SPLINE
SPL {X  -162.820, Y  +438.487, Z    +0.000, E1   -25.409, E3 +468676.662}
SPL {X  -162.820, Y  +441.593, Z    +0.000, E1   -25.391, E3 +468690.270}
SPL {X  -162.820, Y  +444.317, Z    +0.000, E1   -25.492, E3 +468701.452}
SPL {X  -162.820, Y  +446.544, Z    +0.000, E1   -25.427, E3 +468711.621}
SPL {X  -162.820, Y  +448.500, Z    +0.000, E1   -25.425, E3 +468720.223}
SPL {X  -162.820, Y  +451.056, Z    +0.000, E1   -25.443, E3 +468731.330}
SPL {X  -162.820, Y  +454.662, Z    +0.000, E1   -25.474, E3 +468747.074}
SPL {X  -162.820, Y  +458.079, Z    +0.000, E1   -25.369, E3 +468762.654}
SPL {X  -162.820, Y  +460.719, Z    +0.000, E1   -25.411, E3 +468773.912}
SPL {X  -162.820, Y  +463.419, Z    +0.000, E1   -25.510, E3 +468784.949}
SPL {X  -162.820, Y  +466.458, Z    +0.000, E1   -25.433, E3 +468799.005}
SPL {X  -162.820, Y  +470.010, Z    +0.000, E1   -25.445, E3 +468814.373}
SPL {X  -162.820, Y  +472.345, Z    +0.000, E1   -25.448, E3 +468824.460}
SPL {X  -162.820, Y  +475.191, Z    +0.000, E1   -25.489, E3 +468836.822}
SPL {X  -162.820, Y  +478.461, Z    +0.000, E1   -25.410, E3 +468851.592}
SPL {X  -162.820, Y  +480.780, Z    +0.000, E1   -25.447, E3 +468861.453}
SPL {X  -162.820, Y  +483.622, Z    +0.000, E1   -25.381, E3 +468874.495}
SPL {X  -162.820, Y  +487.570, Z    +0.000, E1   -25.482, E3 +468891.133}
SPL {X  -162.820, Y  +491.017, Z    +0.000, E1   -25.445, E3 +468906.348}
SPL {X  -162.820, Y  +494.454, Z    +0.000, E1   -25.465, E3 +468921.407}
SPL {X  -162.820, Y  +498.644, Z    +0.000, E1   -25.463, E3 +468939.784}
SPL {X  -162.820, Y  +502.845, Z    +0.000, E1   -25.458, E3 +468958.217}
SPL {X  -162.820, Y  +506.050, Z    +0.000, E1   -25.420, E3 +468972.357}
SPL {X  -162.820, Y  +508.346, Z    +0.000, E1   -25.444, E3 +468982.205}
SPL {X  -162.820, Y  +511.422, Z    +0.000, E1   -25.445, E3 +468995.865}
SPL {X  -162.820, Y  +515.039, Z    +0.000, E1   -25.452, E3 +469011.547}
SPL {X  -162.820, Y  +518.350, Z    +0.000, E1   -25.425, E3 +469026.296}
SPL {X  -162.820, Y  +521.486, Z    +0.000, E1   -25.382, E3 +469040.324}
SPL {X  -162.820, Y  +524.180, Z    +0.000, E1   -25.495, E3 +469051.196}
SPL {X  -162.820, Y  +527.020, Z    +0.000, E1   -25.477, E3 +469063.889}
SPL {X  -162.820, Y  +530.432, Z    +0.000, E1   -25.477, E3 +469078.755}
SPL {X  -162.820, Y  +534.051, Z    +0.000, E1   -25.484, E3 +469094.632}
SPL {X  -162.820, Y  +537.226, Z    +0.000, E1   -25.378, E3 +469109.201}
SPL {X  -162.820, Y  +539.521, Z    +0.000, E1   -25.386, E3 +469119.160}
SPL {X  -162.820, Y  +542.667, Z    +0.000, E1   -25.474, E3 +469132.485}
SPL {X  -162.820, Y  +546.125, Z    +0.000, E1   -25.505, E3 +469147.210}
SPL {X  -162.820, Y  +549.578, Z    +0.000, E1   -25.462, E3 +469162.834}
SPL {X  -162.820, Y  +553.157, Z    +0.000, E1   -25.443, E3 +469178.497}
SPL {X  -162.820, Y  +556.965, Z    +0.000, E1   -25.478, E3 +469195.090}
SPL {X  -162.820, Y  +561.429, Z    +0.000, E1   -25.478, E3 +469214.608}
SPL {X  -162.820, Y  +565.606, Z    +0.000, E1   -25.468, E3 +469232.939}
SPL {X  -162.820, Y  +568.974, Z    +0.000, E1   -25.453, E3 +469247.649}
SPL {X  -162.820, Y  +572.331, Z    +0.000, E1   -25.489, E3 +469262.198}
SPL {X  -162.820, Y  +576.045, Z    +0.000, E1   -25.412, E3 +469279.006}
SPL {X  -162.820, Y  +580.038, Z    +0.000, E1   -25.473, E3 +469296.101}
SPL {X  -162.820, Y  +583.044, Z    +0.000, E1   -25.450, E3 +469309.224}
SPL {X  -162.820, Y  +585.512, Z    +0.000, E1   -25.448, E3 +469320.120}
SPL {X  -162.820, Y  +588.371, Z    +0.000, E1   -25.460, E3 +469332.506}
SPL {X  -162.820, Y  +591.246, Z    +0.000, E1   -25.415, E3 +469345.525}
SPL {X  -162.820, Y  +594.339, Z    +0.000, E1   -25.487, E3 +469358.428}
SPL {X  -162.820, Y  +596.868, Z    +0.000, E1   -25.461, E3 +469369.691}
SPL {X  -162.820, Y  +600.326, Z    +0.000, E1   -25.438, E3 +469385.212}
SPL {X  -162.820, Y  +604.526, Z    +0.000, E1   -25.502, E3 +469403.035}
SPL {X  -162.820, Y  +607.811, Z    +0.000, E1   -25.507, E3 +469417.250}
SPL {X  -162.820, Y  +611.438, Z    +0.000, E1   -25.467, E3 +469433.610}
SPL {X  -162.820, Y  +615.388, Z    +0.000, E1   -25.455, E3 +469450.869}
SPL {X  -162.820, Y  +618.995, Z    +0.000, E1   -25.483, E3 +469466.464}
SPL {X  -162.820, Y  +622.118, Z    +0.000, E1   -25.492, E3 +469479.929}
SPL {X  -162.820, Y  +624.430, Z    +0.000, E1   -25.475, E3 +469490.150}
SPL {X  -162.820, Y  +626.570, Z    +0.000, E1   -25.441, E3 +469499.751}
SPL {X  -162.820, Y  +628.902, Z    +0.000, E1   -25.449, E3 +469509.931}
SPL {X  -162.820, Y  +631.177, Z    +0.000, E1   -25.467, E3 +469519.762}
SPL {X  -162.820, Y  +633.994, Z    +0.000, E1   -25.503, E3 +469531.809}
SPL {X  -162.820, Y  +636.469, Z    +0.000, E1   -25.465, E3 +469542.852}
SPL {X  -162.820, Y  +638.486, Z    +0.000, E1   -25.456, E3 +469551.770}
SPL {X  -162.820, Y  +640.803, Z    +0.000, E1   -25.462, E3 +469561.831}
SPL {X  -162.820, Y  +643.028, Z    +0.000, E1   -25.494, E3 +469571.341}
SPL {X  -162.820, Y  +646.519, Z    +0.000, E1   -25.551, E3 +469586.323}
SPL {X  -162.820, Y  +649.837, Z    +0.000, E1   -25.446, E3 +469601.447}
SPL {X  -162.820, Y  +652.810, Z    +0.000, E1   -25.497, E3 +469614.090}
SPL {X  -162.820, Y  +655.214, Z    +0.000, E1   -25.485, E3 +469624.593}
SPL {X  -162.820, Y  +657.616, Z    +0.000, E1   -25.511, E3 +469634.947}
SPL {X  -162.820, Y  +660.007, Z    +0.000, E1   -25.550, E3 +469645.008}
SPL {X  -162.820, Y  +662.980, Z    +0.000, E1   -25.505, E3 +469658.567}
SPL {X  -162.820, Y  +667.253, Z    +0.000, E1   -25.483, E3 +469677.443}
SPL {X  -162.820, Y  +671.102, Z    +0.000, E1   -25.514, E3 +469693.894}
SPL {X  -162.820, Y  +673.648, Z    +0.000, E1   -25.431, E3 +469705.560}
SPL {X  -162.796, Y  +676.319, Z    +0.000, E1   -25.526, E3 +469716.570}
SPL {X  -162.707, Y  +679.552, Z    +0.000, E1   -25.443, E3 +469731.445}
SPL {X  -162.545, Y  +682.952, Z    +0.000, E1   -25.510, E3 +469745.678}
SPL {X  -162.381, Y  +685.455, Z    +0.000, E1   -25.410, E3 +469757.364}
SPL {X  -162.194, Y  +687.760, Z    +0.000, E1   -25.360, E3 +469767.800}
SPL {X  -161.866, Y  +691.104, Z    +0.000, E1   -25.383, E3 +469782.432}
SPL {X  -161.319, Y  +695.558, Z    +0.000, E1   -25.832, E3 +469798.234}
SPL {X  -157.976, Y  +712.921, Z    +0.000, E1   -33.197, E3 +469811.626}
ENDSPLINE

SPLINE
SPL {X  -160.738, Y  +699.453, Z    +0.000, E1   -21.994, E3 +469849.253}
SPL {X  -161.689, Y  +692.657, Z    +0.000, E1   -15.656, E3 +469889.323}
SPL {X  -162.807, Y  +675.545, Z    +0.000, E1    -5.787, E3 +469884.822}
ENDSPLINE

SPLINE
SPL {X  -162.791, Y  +676.574, Z    +0.000, E1    -6.127, E3 +469897.925}
ENDSPLINE

SPLINE
SPL {X  -162.820, Y  +664.716, Z    +0.000, E1    +1.705, E3 +469886.799}
SPL {X  -162.820, Y  +658.484, Z    +0.000, E1    +6.336, E3 +469893.276}
SPL {X  -162.820, Y  +640.102, Z    +0.000, E1   +22.409, E3 +469888.014}
SPL {X  -162.820, Y  +633.503, Z    +0.000, E1   +21.975, E3 +469920.251}
SPL {X  -162.820, Y  +611.299, Z    +0.000, E1   +31.088, E3 +469948.363}
ENDSPLINE

SPLINE
SPL {X  -162.820, Y  +618.877, Z    +0.000, E1   +25.259, E3 +469959.858}
ENDSPLINE

SPLINE
SPL {X  -162.820, Y  +617.582, Z    +0.000, E1   +24.552, E3 +469971.235}
SPL {X  -162.820, Y  +614.716, Z    +0.000, E1   +24.535, E3 +469984.446}
SPL {X  -162.820, Y  +611.754, Z    +0.000, E1   +24.563, E3 +469997.734}
SPL {X  -162.820, Y  +608.970, Z    +0.000, E1   +24.542, E3 +470010.574}
SPL {X  -162.820, Y  +606.285, Z    +0.000, E1   +24.533, E3 +470022.910}
SPL {X  -162.820, Y  +603.509, Z    +0.000, E1   +24.546, E3 +470035.447}
SPL {X  -162.820, Y  +600.818, Z    +0.000, E1   +24.590, E3 +470047.370}
SPL {X  -162.820, Y  +598.053, Z    +0.000, E1   +24.547, E3 +470060.353}
SPL {X  -162.820, Y  +595.188, Z    +0.000, E1   +24.538, E3 +470073.441}
SPL {X  -162.820, Y  +592.738, Z    +0.000, E1   +24.551, E3 +470084.490}
SPL {X  -162.820, Y  +590.118, Z    +0.000, E1   +24.544, E3 +470096.549}
SPL {X  -162.820, Y  +587.204, Z    +0.000, E1   +24.592, E3 +470109.426}
SPL {X  -162.820, Y  +584.766, Z    +0.000, E1   +24.499, E3 +470121.259}
SPL {X  -162.820, Y  +581.896, Z    +0.000, E1   +24.528, E3 +470134.201}
SPL {X  -162.820, Y  +579.244, Z    +0.000, E1   +24.610, E3 +470145.545}
SPL {X  -162.820, Y  +576.848, Z    +0.000, E1   +24.543, E3 +470157.086}
SPL {X  -162.820, Y  +573.694, Z    +0.000, E1   +24.535, E3 +470171.556}
SPL {X  -162.820, Y  +570.310, Z    +0.000, E1   +24.556, E3 +470186.872}
SPL {X  -162.820, Y  +567.494, Z    +0.000, E1   +24.547, E3 +470199.657}
SPL {X  -162.820, Y  +564.977, Z    +0.000, E1   +24.571, E3 +470210.987}
SPL {X  -162.820, Y  +562.356, Z    +0.000, E1   +24.575, E3 +470222.886}
SPL {X  -162.820, Y  +558.990, Z    +0.000, E1   +24.558, E3 +470238.536}
SPL {X  -162.820, Y  +555.584, Z    +0.000, E1   +24.559, E3 +470253.905}
SPL {X  -162.820, Y  +552.169, Z    +0.000, E1   +24.581, E3 +470269.474}
SPL {X  -162.820, Y  +548.172, Z    +0.000, E1   +24.564, E3 +470287.822}
SPL {X  -162.820, Y  +544.025, Z    +0.000, E1   +24.611, E3 +470306.376}
SPL {X  -162.820, Y  +540.573, Z    +0.000, E1   +24.503, E3 +470322.830}
SPL {X  -162.820, Y  +537.211, Z    +0.000, E1   +24.561, E3 +470337.759}
SPL {X  -162.820, Y  +534.025, Z    +0.000, E1   +24.589, E3 +470352.003}
SPL {X  -162.820, Y  +531.527, Z    +0.000, E1   +24.582, E3 +470363.388}
SPL {X  -162.820, Y  +529.165, Z    +0.000, E1   +24.521, E3 +470374.637}
SPL {X  -162.820, Y  +525.802, Z    +0.000, E1   +24.585, E3 +470389.657}
SPL {X  -162.820, Y  +521.731, Z    +0.000, E1   +24.542, E3 +470408.593}
SPL {X  -162.820, Y  +518.185, Z    +0.000, E1   +24.561, E3 +470424.465}
SPL {X  -162.820, Y  +508.728, Z    +0.000, E1   +28.484, E3 +470435.005}
SPL {X  -162.820, Y  +500.664, Z    +0.000, E1   +31.476, E3 +470443.669}
SPL {X  -162.820, Y  +499.290, Z    +0.000, E1   +30.657, E3 +470453.951}
SPL {X  -162.820, Y  +497.700, Z    +0.000, E1   +29.785, E3 +470465.566}
SPL {X  -162.820, Y  +495.915, Z    +0.000, E1   +28.861, E3 +470478.658}
SPL {X  -162.820, Y  +494.678, Z    +0.000, E1   +27.647, E3 +470492.004}
SPL {X  -162.820, Y  +493.757, Z    +0.000, E1   +26.462, E3 +470504.364}
SPL {X  -162.820, Y  +492.330, Z    +0.000, E1   +25.953, E3 +470514.118}
SPL {X  -162.820, Y  +489.800, Z    +0.000, E1   +25.653, E3 +470527.580}
SPL {X  -162.820, Y  +485.392, Z    +0.000, E1   +25.667, E3 +470546.607}
SPL {X  -162.820, Y  +482.092, Z    +0.000, E1   +25.593, E3 +470561.295}
SPL {X  -162.820, Y  +479.578, Z    +0.000, E1   +25.634, E3 +470571.938}
SPL {X  -162.820, Y  +477.137, Z    +0.000, E1   +25.632, E3 +470582.517}
SPL {X  -162.820, Y  +473.770, Z    +0.000, E1   +25.664, E3 +470597.063}
SPL {X  -162.820, Y  +469.694, Z    +0.000, E1   +25.657, E3 +470614.794}
SPL {X  -162.820, Y  +465.727, Z    +0.000, E1   +25.676, E3 +470631.837}
SPL {X  -162.820, Y  +461.675, Z    +0.000, E1   +25.655, E3 +470649.643}
SPL {X  -162.820, Y  +457.479, Z    +0.000, E1   +25.656, E3 +470667.823}
SPL {X  -162.820, Y  +453.678, Z    +0.000, E1   +25.652, E3 +470684.275}
SPL {X  -162.820, Y  +450.466, Z    +0.000, E1   +25.644, E3 +470698.220}
SPL {X  -162.820, Y  +447.822, Z    +0.000, E1   +25.664, E3 +470709.478}
SPL {X  -162.820, Y  +445.556, Z    +0.000, E1   +25.626, E3 +470719.609}
SPL {X  -162.820, Y  +442.508, Z    +0.000, E1   +25.657, E3 +470732.703}
SPL {X  -162.820, Y  +439.273, Z    +0.000, E1   +25.576, E3 +470747.341}
SPL {X  -162.820, Y  +435.635, Z    +0.000, E1   +25.661, E3 +470762.572}
SPL {X  -162.820, Y  +431.823, Z    +0.000, E1   +25.651, E3 +470779.221}
SPL {X  -162.820, Y  +427.740, Z    +0.000, E1   +25.667, E3 +470796.849}
SPL {X  -162.820, Y  +423.655, Z    +0.000, E1   +25.628, E3 +470814.874}
SPL {X  -162.820, Y  +419.407, Z    +0.000, E1   +25.665, E3 +470833.066}
SPL {X  -162.820, Y  +415.900, Z    +0.000, E1   +25.638, E3 +470848.335}
SPL {X  -162.820, Y  +412.302, Z    +0.000, E1   +25.662, E3 +470863.947}
SPL {X  -162.820, Y  +408.133, Z    +0.000, E1   +25.637, E3 +470882.205}
SPL {X  -162.820, Y  +404.293, Z    +0.000, E1   +25.628, E3 +470898.928}
SPL {X  -162.820, Y  +400.835, Z    +0.000, E1   +25.694, E3 +470913.327}
SPL {X  -162.820, Y  +398.703, Z    +0.000, E1   +25.586, E3 +470923.319}
SPL {X  -162.820, Y  +395.582, Z    +0.000, E1   +25.684, E3 +470936.311}
SPL {X  -162.820, Y  +391.417, Z    +0.000, E1   +25.659, E3 +470954.649}
SPL {X  -162.820, Y  +387.939, Z    +0.000, E1   +25.627, E3 +470969.796}
SPL {X  -162.820, Y  +384.398, Z    +0.000, E1   +25.707, E3 +470984.694}
SPL {X  -162.820, Y  +380.448, Z    +0.000, E1   +25.674, E3 +471002.057}
SPL {X  -162.785, Y  +377.106, Z    +0.000, E1   +25.598, E3 +471017.001}
SPL {X  -162.663, Y  +373.346, Z    +0.000, E1   +25.707, E3 +471032.652}
SPL {X  -162.487, Y  +370.088, Z    +0.000, E1   +25.525, E3 +471047.987}
SPL {X  -162.307, Y  +367.587, Z    +0.000, E1   +25.577, E3 +471058.405}
SPL {X  -162.041, Y  +364.588, Z    +0.000, E1   +25.591, E3 +471071.483}
SPL {X  -161.760, Y  +361.954, Z    +0.000, E1   +25.495, E3 +471083.430}
SPL {X  -161.454, Y  +359.455, Z    +0.000, E1   +25.428, E3 +471094.905}
SPL {X  -160.939, Y  +355.820, Z    +0.000, E1   +26.179, E3 +471104.788}
SPL {X  -155.035, Y  +330.756, Z    +0.000, E1   +37.918, E3 +471111.121}
SPL {X  -153.918, Y  +327.401, Z    +0.000, E1   +34.677, E3 +471146.422}
ENDSPLINE

SPLINE
SPL {X  -159.701, Y  +348.785, Z    +0.000, E1   +24.361, E3 +471153.903}
SPL {X  -162.442, Y  +369.407, Z    +0.000, E1   +11.234, E3 +471183.538}
SPL {X  -162.820, Y  +384.333, Z    +0.000, E1    +1.902, E3 +471184.744}
SPL {X  -162.820, Y  +389.940, Z    +0.000, E1    -2.281, E3 +471187.666}
SPL {X  -162.820, Y  +396.652, Z    +0.000, E1    -7.520, E3 +471187.244}
SPL {X  -162.820, Y  +406.605, Z    +0.000, E1   -16.760, E3 +471179.721}
SPL {X  -162.820, Y  +418.675, Z    +0.000, E1   -22.201, E3 +471205.970}
SPL {X  -162.820, Y  +425.113, Z    +0.000, E1   -25.243, E3 +471214.906}
SPL {X  -162.820, Y  +441.937, Z    +0.000, E1   -31.578, E3 +471236.984}
ENDSPLINE

SPLINE
SPL {X  -162.820, Y  +437.771, Z    +0.000, E1   -26.555, E3 +471256.084}
ENDSPLINE

SPLINE
SPL {X  -162.820, Y  +439.120, Z    +0.000, E1   -25.352, E3 +471270.628}
SPL {X  -162.820, Y  +441.593, Z    +0.000, E1   -25.391, E3 +471281.179}
SPL {X  -162.820, Y  +444.317, Z    +0.000, E1   -25.492, E3 +471292.361}
SPL {X  -162.820, Y  +446.544, Z    +0.000, E1   -25.427, E3 +471302.530}
SPL {X  -162.820, Y  +448.500, Z    +0.000, E1   -25.425, E3 +471311.132}
SPL {X  -162.820, Y  +451.056, Z    +0.000, E1   -25.443, E3 +471322.239}
SPL {X  -162.820, Y  +454.662, Z    +0.000, E1   -25.474, E3 +471337.984}
SPL {X  -162.820, Y  +458.079, Z    +0.000, E1   -25.369, E3 +471353.563}
SPL {X  -162.820, Y  +460.719, Z    +0.000, E1   -25.411, E3 +471364.821}
SPL {X  -162.820, Y  +463.419, Z    +0.000, E1   -25.510, E3 +471375.859}
SPL {X  -162.820, Y  +465.376, Z    +0.000, E1   -25.372, E3 +471385.446}
SPL {X  -162.820, Y  +467.440, Z    +0.000, E1   -25.427, E3 +471394.078}
SPL {X  -162.820, Y  +470.010, Z    +0.000, E1   -25.445, E3 +471405.283}
SPL {X  -162.820, Y  +473.445, Z    +0.000, E1   -25.493, E3 +471420.006}
SPL {X  -162.820, Y  +476.157, Z    +0.000, E1   -25.426, E3 +471432.221}
SPL {X  -162.820, Y  +478.461, Z    +0.000, E1   -25.410, E3 +471442.501}
SPL {X  -162.820, Y  +481.644, Z    +0.000, E1   -25.433, E3 +471456.447}
SPL {X  -162.820, Y  +486.042, Z    +0.000, E1   -25.483, E3 +471475.367}
SPL {X  -162.820, Y  +490.287, Z    +0.000, E1   -25.463, E3 +471494.085}
SPL {X  -162.820, Y  +494.454, Z    +0.000, E1   -25.465, E3 +471512.316}
SPL {X  -162.820, Y  +498.644, Z    +0.000, E1   -25.463, E3 +471530.693}
SPL {X  -162.820, Y  +502.845, Z    +0.000, E1   -25.458, E3 +471549.126}
SPL {X  -162.820, Y  +506.050, Z    +0.000, E1   -25.420, E3 +471563.266}
SPL {X  -162.820, Y  +508.346, Z    +0.000, E1   -25.444, E3 +471573.114}
SPL {X  -162.820, Y  +511.422, Z    +0.000, E1   -25.445, E3 +471586.775}
SPL {X  -162.820, Y  +515.039, Z    +0.000, E1   -25.452, E3 +471602.456}
SPL {X  -162.820, Y  +517.481, Z    +0.000, E1   -25.432, E3 +471613.190}
SPL {X  -162.820, Y  +519.134, Z    +0.000, E1   -25.366, E3 +471620.937}
SPL {X  -162.820, Y  +521.486, Z    +0.000, E1   -25.382, E3 +471631.233}
SPL {X  -162.820, Y  +525.073, Z    +0.000, E1   -25.512, E3 +471646.039}
SPL {X  -162.820, Y  +528.658, Z    +0.000, E1   -25.482, E3 +471661.924}
SPL {X  -162.820, Y  +532.006, Z    +0.000, E1   -25.455, E3 +471676.713}
SPL {X  -162.820, Y  +534.806, Z    +0.000, E1   -25.465, E3 +471688.829}
SPL {X  -162.820, Y  +537.226, Z    +0.000, E1   -25.378, E3 +471700.111}
SPL {X  -162.820, Y  +540.345, Z    +0.000, E1   -25.451, E3 +471713.292}
SPL {X  -162.820, Y  +543.279, Z    +0.000, E1   -25.419, E3 +471726.324}
SPL {X  -162.820, Y  +546.125, Z    +0.000, E1   -25.505, E3 +471738.119}
SPL {X  -162.820, Y  +549.578, Z    +0.000, E1   -25.462, E3 +471753.743}
SPL {X  -162.820, Y  +553.157, Z    +0.000, E1   -25.443, E3 +471769.407}
SPL {X  -162.820, Y  +556.965, Z    +0.000, E1   -25.478, E3 +471785.999}
SPL {X  -162.820, Y  +561.429, Z    +0.000, E1   -25.478, E3 +471805.518}
SPL {X  -162.820, Y  +565.606, Z    +0.000, E1   -25.468, E3 +471823.848}
SPL {X  -162.820, Y  +568.974, Z    +0.000, E1   -25.453, E3 +471838.558}
SPL {X  -162.820, Y  +571.303, Z    +0.000, E1   -25.427, E3 +471848.905}
SPL {X  -162.820, Y  +574.067, Z    +0.000, E1   -25.459, E3 +471860.844}
SPL {X  -162.820, Y  +576.597, Z    +0.000, E1   -25.400, E3 +471872.315}
SPL {X  -162.820, Y  +578.977, Z    +0.000, E1   -25.460, E3 +471882.247}
SPL {X  -162.820, Y  +581.995, Z    +0.000, E1   -25.468, E3 +471895.606}
SPL {X  -162.820, Y  +585.512, Z    +0.000, E1   -25.448, E3 +471911.029}
SPL {X  -162.820, Y  +588.371, Z    +0.000, E1   -25.460, E3 +471923.415}
SPL {X  -162.820, Y  +591.246, Z    +0.000, E1   -25.415, E3 +471936.434}
SPL {X  -162.820, Y  +594.339, Z    +0.000, E1   -25.487, E3 +471949.337}
SPL {X  -162.820, Y  +596.868, Z    +0.000, E1   -25.461, E3 +471960.600}
SPL {X  -162.820, Y  +600.326, Z    +0.000, E1   -25.438, E3 +471976.121}
SPL {X  -162.820, Y  +604.526, Z    +0.000, E1   -25.502, E3 +471993.944}
SPL {X  -162.820, Y  +607.811, Z    +0.000, E1   -25.507, E3 +472008.159}
SPL {X  -162.820, Y  +611.438, Z    +0.000, E1   -25.467, E3 +472024.519}
SPL {X  -162.820, Y  +615.388, Z    +0.000, E1   -25.455, E3 +472041.778}
SPL {X  -162.820, Y  +618.995, Z    +0.000, E1   -25.483, E3 +472057.373}
SPL {X  -162.820, Y  +622.118, Z    +0.000, E1   -25.492, E3 +472070.838}
SPL {X  -162.820, Y  +624.430, Z    +0.000, E1   -25.475, E3 +472081.059}
SPL {X  -162.820, Y  +626.570, Z    +0.000, E1   -25.441, E3 +472090.660}
SPL {X  -162.820, Y  +628.902, Z    +0.000, E1   -25.449, E3 +472100.840}
SPL {X  -162.820, Y  +631.177, Z    +0.000, E1   -25.467, E3 +472110.671}
SPL {X  -162.820, Y  +633.994, Z    +0.000, E1   -25.503, E3 +472122.718}
SPL {X  -162.820, Y  +636.469, Z    +0.000, E1   -25.465, E3 +472133.761}
SPL {X  -162.820, Y  +638.486, Z    +0.000, E1   -25.456, E3 +472142.679}
SPL {X  -162.820, Y  +640.803, Z    +0.000, E1   -25.462, E3 +472152.740}
SPL {X  -162.820, Y  +643.028, Z    +0.000, E1   -25.494, E3 +472162.250}
SPL {X  -162.820, Y  +645.694, Z    +0.000, E1   -25.540, E3 +472173.537}
SPL {X  -162.820, Y  +649.102, Z    +0.000, E1   -25.495, E3 +472188.965}
SPL {X  -162.820, Y  +652.810, Z    +0.000, E1   -25.497, E3 +472204.999}
SPL {X  -162.820, Y  +655.214, Z    +0.000, E1   -25.485, E3 +472215.502}
SPL {X  -162.820, Y  +657.616, Z    +0.000, E1   -25.511, E3 +472225.856}
SPL {X  -162.820, Y  +660.851, Z    +0.000, E1   -25.520, E3 +472239.999}
SPL {X  -162.820, Y  +663.853, Z    +0.000, E1   -25.496, E3 +472253.180}
SPL {X  -162.820, Y  +666.096, Z    +0.000, E1   -25.408, E3 +472263.647}
SPL {X  -162.820, Y  +669.195, Z    +0.000, E1   -25.525, E3 +472276.484}
SPL {X  -162.820, Y  +672.979, Z    +0.000, E1   -25.478, E3 +472293.334}
SPL {X  -162.796, Y  +676.319, Z    +0.000, E1   -25.526, E3 +472307.479}
SPL {X  -162.739, Y  +678.625, Z    +0.000, E1   -25.423, E3 +472318.271}
SPL {X  -162.669, Y  +680.515, Z    +0.000, E1   -25.398, E3 +472326.725}
SPL {X  -162.545, Y  +682.952, Z    +0.000, E1   -25.510, E3 +472336.587}
SPL {X  -162.381, Y  +685.455, Z    +0.000, E1   -25.410, E3 +472348.273}
SPL {X  -162.194, Y  +687.760, Z    +0.000, E1   -25.360, E3 +472358.709}
SPL {X  -161.866, Y  +691.104, Z    +0.000, E1   -25.383, E3 +472373.341}
SPL {X  -161.024, Y  +697.619, Z    +0.000, E1   -26.780, E3 +472390.572}
SPL {X  -157.189, Y  +715.948, Z    +0.000, E1   -34.218, E3 +472405.491}
ENDSPLINE

SPLINE
SPL {X  -157.848, Y  +713.428, Z    +0.000, E1   -28.857, E3 +472439.630}
SPL {X  -161.035, Y  +697.541, Z    +0.000, E1   -20.899, E3 +472440.149}
SPL {X  -161.689, Y  +692.657, Z    +0.000, E1   -15.656, E3 +472480.232}
SPL {X  -162.807, Y  +675.545, Z    +0.000, E1    -5.787, E3 +472475.732}
ENDSPLINE

SPLINE
SPL {X  -162.791, Y  +676.574, Z    +0.000, E1    -6.127, E3 +472488.834}
ENDSPLINE

SPLINE
SPL {X  -162.820, Y  +664.716, Z    +0.000, E1    +1.705, E3 +472477.708}
SPL {X  -162.820, Y  +658.484, Z    +0.000, E1    +6.336, E3 +472484.185}
SPL {X  -162.820, Y  +640.102, Z    +0.000, E1   +22.409, E3 +472478.923}
SPL {X  -162.820, Y  +633.503, Z    +0.000, E1   +21.975, E3 +472511.160}
SPL {X  -162.820, Y  +611.299, Z    +0.000, E1   +31.088, E3 +472539.273}
ENDSPLINE

SPLINE
SPL {X  -162.820, Y  +618.877, Z    +0.000, E1   +25.259, E3 +472550.767}
ENDSPLINE

SPLINE
SPL {X  -162.820, Y  +617.582, Z    +0.000, E1   +24.552, E3 +472562.144}
SPL {X  -162.820, Y  +614.716, Z    +0.000, E1   +24.535, E3 +472575.355}
SPL {X  -162.820, Y  +611.754, Z    +0.000, E1   +24.563, E3 +472588.643}
SPL {X  -162.820, Y  +608.970, Z    +0.000, E1   +24.542, E3 +472601.483}
SPL {X  -162.820, Y  +606.285, Z    +0.000, E1   +24.533, E3 +472613.819}
SPL {X  -162.820, Y  +603.509, Z    +0.000, E1   +24.546, E3 +472626.356}
SPL {X  -162.820, Y  +600.230, Z    +0.000, E1   +24.589, E3 +472641.101}
SPL {X  -162.820, Y  +597.446, Z    +0.000, E1   +24.542, E3 +472653.960}
SPL {X  -162.820, Y  +595.188, Z    +0.000, E1   +24.538, E3 +472664.351}
SPL {X  -162.820, Y  +592.738, Z    +0.000, E1   +24.551, E3 +472675.399}
SPL {X  -162.820, Y  +590.118, Z    +0.000, E1   +24.544, E3 +472687.458}
SPL {X  -162.820, Y  +587.204, Z    +0.000, E1   +24.592, E3 +472700.335}
SPL {X  -162.820, Y  +584.766, Z    +0.000, E1   +24.499, E3 +472712.168}
SPL {X  -162.820, Y  +581.896, Z    +0.000, E1   +24.528, E3 +472725.110}
SPL {X  -162.820, Y  +579.244, Z    +0.000, E1   +24.610, E3 +472736.454}
SPL {X  -162.820, Y  +576.848, Z    +0.000, E1   +24.543, E3 +472747.995}
SPL {X  -162.820, Y  +574.433, Z    +0.000, E1   +24.551, E3 +472758.826}
SPL {X  -162.820, Y  +572.074, Z    +0.000, E1   +24.505, E3 +472770.097}
SPL {X  -162.820, Y  +569.438, Z    +0.000, E1   +24.562, E3 +472781.556}
SPL {X  -162.820, Y  +567.494, Z    +0.000, E1   +24.547, E3 +472790.566}
SPL {X  -162.820, Y  +564.977, Z    +0.000, E1   +24.571, E3 +472801.896}
SPL {X  -162.820, Y  +562.356, Z    +0.000, E1   +24.575, E3 +472813.795}
SPL {X  -162.820, Y  +560.119, Z    +0.000, E1   +24.506, E3 +472824.484}
SPL {X  -162.820, Y  +558.093, Z    +0.000, E1   +24.537, E3 +472833.502}
SPL {X  -162.820, Y  +555.584, Z    +0.000, E1   +24.559, E3 +472844.814}
SPL {X  -162.820, Y  +552.169, Z    +0.000, E1   +24.581, E3 +472860.383}
SPL {X  -162.820, Y  +548.172, Z    +0.000, E1   +24.564, E3 +472878.731}
SPL {X  -162.820, Y  +544.025, Z    +0.000, E1   +24.611, E3 +472897.285}
SPL {X  -162.820, Y  +540.573, Z    +0.000, E1   +24.503, E3 +472913.739}
SPL {X  -162.820, Y  +538.106, Z    +0.000, E1   +24.553, E3 +472924.493}
SPL {X  -162.820, Y  +536.451, Z    +0.000, E1   +24.519, E3 +472932.311}
SPL {X  -162.820, Y  +534.025, Z    +0.000, E1   +24.589, E3 +472942.912}
SPL {X  -162.820, Y  +531.527, Z    +0.000, E1   +24.582, E3 +472954.297}
SPL {X  -162.820, Y  +529.165, Z    +0.000, E1   +24.521, E3 +472965.546}
SPL {X  -162.820, Y  +526.822, Z    +0.000, E1   +24.559, E3 +472975.909}
SPL {X  -162.820, Y  +524.112, Z    +0.000, E1   +24.542, E3 +472988.527}
SPL {X  -162.820, Y  +521.048, Z    +0.000, E1   +24.515, E3 +473002.663}
SPL {X  -162.820, Y  +518.185, Z    +0.000, E1   +24.561, E3 +473015.374}
SPL {X  -162.820, Y  +508.728, Z    +0.000, E1   +28.484, E3 +473025.914}
SPL {X  -162.820, Y  +500.664, Z    +0.000, E1   +31.476, E3 +473034.578}
SPL {X  -162.820, Y  +499.290, Z    +0.000, E1   +30.657, E3 +473044.860}
SPL {X  -162.820, Y  +497.700, Z    +0.000, E1   +29.785, E3 +473056.475}
SPL {X  -162.820, Y  +495.915, Z    +0.000, E1   +28.861, E3 +473069.567}
SPL {X  -162.820, Y  +494.678, Z    +0.000, E1   +27.647, E3 +473082.913}
SPL {X  -162.820, Y  +493.757, Z    +0.000, E1   +26.462, E3 +473095.273}
SPL {X  -162.820, Y  +491.420, Z    +0.000, E1   +25.780, E3 +473110.534}
SPL {X  -162.820, Y  +488.594, Z    +0.000, E1   +25.642, E3 +473123.574}
SPL {X  -162.820, Y  +485.392, Z    +0.000, E1   +25.667, E3 +473137.516}
SPL {X  -162.820, Y  +482.092, Z    +0.000, E1   +25.593, E3 +473152.204}
SPL {X  -162.820, Y  +479.578, Z    +0.000, E1   +25.634, E3 +473162.847}
SPL {X  -162.820, Y  +476.226, Z    +0.000, E1   +25.672, E3 +473177.237}
SPL {X  -162.820, Y  +473.037, Z    +0.000, E1   +25.618, E3 +473191.328}
SPL {X  -162.820, Y  +469.694, Z    +0.000, E1   +25.657, E3 +473205.703}
SPL {X  -162.820, Y  +465.727, Z    +0.000, E1   +25.676, E3 +473222.746}
SPL {X  -162.820, Y  +463.001, Z    +0.000, E1   +25.614, E3 +473234.862}
SPL {X  -162.820, Y  +459.882, Z    +0.000, E1   +25.674, E3 +473248.163}
SPL {X  -162.820, Y  +456.773, Z    +0.000, E1   +25.591, E3 +473262.109}
SPL {X  -162.820, Y  +454.429, Z    +0.000, E1   +25.642, E3 +473271.877}
SPL {X  -162.820, Y  +451.204, Z    +0.000, E1   +25.672, E3 +473285.903}
SPL {X  -162.820, Y  +447.822, Z    +0.000, E1   +25.664, E3 +473300.387}
SPL {X  -162.820, Y  +445.556, Z    +0.000, E1   +25.626, E3 +473310.518}
SPL {X  -162.820, Y  +442.508, Z    +0.000, E1   +25.657, E3 +473323.612}
SPL {X  -162.820, Y  +439.273, Z    +0.000, E1   +25.576, E3 +473338.250}
SPL {X  -162.820, Y  +436.773, Z    +0.000, E1   +25.602, E3 +473348.814}
SPL {X  -162.820, Y  +434.768, Z    +0.000, E1   +25.655, E3 +473357.131}
SPL {X  -162.820, Y  +431.823, Z    +0.000, E1   +25.651, E3 +473370.130}
SPL {X  -162.820, Y  +427.740, Z    +0.000, E1   +25.667, E3 +473387.759}
SPL {X  -162.820, Y  +423.655, Z    +0.000, E1   +25.628, E3 +473405.783}
SPL {X  -162.820, Y  +419.407, Z    +0.000, E1   +25.665, E3 +473423.975}
SPL {X  -162.820, Y  +415.900, Z    +0.000, E1   +25.638, E3 +473439.245}
SPL {X  -162.820, Y  +413.088, Z    +0.000, E1   +25.644, E3 +473451.401}
SPL {X  -162.820, Y  +410.320, Z    +0.000, E1   +25.604, E3 +473463.720}
SPL {X  -162.820, Y  +407.487, Z    +0.000, E1   +25.617, E3 +473475.927}
SPL {X  -162.820, Y  +405.108, Z    +0.000, E1   +25.535, E3 +473486.895}
SPL {X  -162.820, Y  +401.373, Z    +0.000, E1   +25.736, E3 +473501.732}
SPL {X  -162.820, Y  +398.703, Z    +0.000, E1   +25.586, E3 +473514.228}
SPL {X  -162.820, Y  +395.582, Z    +0.000, E1   +25.684, E3 +473527.220}
SPL {X  -162.820, Y  +391.417, Z    +0.000, E1   +25.659, E3 +473545.558}
SPL {X  -162.820, Y  +387.939, Z    +0.000, E1   +25.627, E3 +473560.705}
SPL {X  -162.820, Y  +385.565, Z    +0.000, E1   +25.686, E3 +473570.494}
SPL {X  -162.820, Y  +383.458, Z    +0.000, E1   +25.657, E3 +473579.858}
SPL {X  -162.820, Y  +381.229, Z    +0.000, E1   +25.660, E3 +473589.533}
SPL {X  -162.797, Y  +377.786, Z    +0.000, E1   +25.638, E3 +473604.823}
SPL {X  -162.663, Y  +373.346, Z    +0.000, E1   +25.707, E3 +473623.561}
SPL {X  -162.487, Y  +370.088, Z    +0.000, E1   +25.525, E3 +473638.896}
SPL {X  -162.307, Y  +367.587, Z    +0.000, E1   +25.577, E3 +473649.314}
SPL {X  -162.041, Y  +364.588, Z    +0.000, E1   +25.591, E3 +473662.392}
SPL {X  -161.695, Y  +361.389, Z    +0.000, E1   +25.445, E3 +473677.278}
SPL {X  -161.190, Y  +357.520, Z    +0.000, E1   +25.774, E3 +473691.529}
SPL {X  -155.035, Y  +330.756, Z    +0.000, E1   +37.918, E3 +473702.031}
SPL {X  -153.918, Y  +327.401, Z    +0.000, E1   +34.677, E3 +473737.331}
ENDSPLINE

SPLINE
SPL {X  -159.701, Y  +348.785, Z    +0.000, E1   +24.361, E3 +473744.812}
SPL {X  -162.442, Y  +369.407, Z    +0.000, E1   +11.234, E3 +473774.447}
SPL {X  -162.820, Y  +384.333, Z    +0.000, E1    +1.902, E3 +473775.653}
SPL {X  -162.820, Y  +389.940, Z    +0.000, E1    -2.281, E3 +473778.575}
SPL {X  -162.820, Y  +396.652, Z    +0.000, E1    -7.520, E3 +473778.153}
SPL {X  -162.820, Y  +406.605, Z    +0.000, E1   -16.760, E3 +473770.630}
SPL {X  -162.820, Y  +420.013, Z    +0.000, E1   -22.833, E3 +473798.751}
SPL {X  -162.820, Y  +442.075, Z    +0.000, E1   -31.090, E3 +473831.537}
ENDSPLINE

SPLINE
SPL {X  -162.820, Y  +436.680, Z    +0.000, E1   -26.151, E3 +473844.841}
ENDSPLINE

SPLINE
SPL {X  -162.820, Y  +438.487, Z    +0.000, E1   -25.409, E3 +473858.480}
SPL {X  -162.820, Y  +441.593, Z    +0.000, E1   -25.391, E3 +473872.088}
SPL {X  -162.820, Y  +444.317, Z    +0.000, E1   -25.492, E3 +473883.270}
SPL {X  -162.820, Y  +447.641, Z    +0.000, E1   -25.460, E3 +473898.205}
SPL {X  -162.820, Y  +451.056, Z    +0.000, E1   -25.443, E3 +473913.148}
SPL {X  -162.820, Y  +454.662, Z    +0.000, E1   -25.474, E3 +473928.893}
SPL {X  -162.820, Y  +458.079, Z    +0.000, E1   -25.369, E3 +473944.472}
SPL {X  -162.820, Y  +460.719, Z    +0.000, E1   -25.411, E3 +473955.730}
SPL {X  -162.820, Y  +463.419, Z    +0.000, E1   -25.510, E3 +473966.768}
SPL {X  -162.820, Y  +465.376, Z    +0.000, E1   -25.372, E3 +473976.355}
SPL {X  -162.820, Y  +467.440, Z    +0.000, E1   -25.427, E3 +473984.987}
SPL {X  -162.820, Y  +470.010, Z    +0.000, E1   -25.445, E3 +473996.192}
SPL {X  -162.820, Y  +473.445, Z    +0.000, E1   -25.493, E3 +474010.915}
SPL {X  -162.820, Y  +476.157, Z    +0.000, E1   -25.426, E3 +474023.130}
SPL {X  -162.820, Y  +478.461, Z    +0.000, E1   -25.410, E3 +474033.410}
SPL {X  -162.820, Y  +481.644, Z    +0.000, E1   -25.433, E3 +474047.357}
SPL {X  -162.820, Y  +486.042, Z    +0.000, E1   -25.483, E3 +474066.276}
SPL {X  -162.820, Y  +490.287, Z    +0.000, E1   -25.463, E3 +474084.994}
SPL {X  -162.820, Y  +494.454, Z    +0.000, E1   -25.465, E3 +474103.225}
SPL {X  -162.820, Y  +498.644, Z    +0.000, E1   -25.463, E3 +474121.602}
SPL {X  -162.820, Y  +502.003, Z    +0.000, E1   -25.416, E3 +474136.499}
SPL {X  -162.820, Y  +505.370, Z    +0.000, E1   -25.456, E3 +474151.075}
SPL {X  -162.820, Y  +509.412, Z    +0.000, E1   -25.458, E3 +474168.798}
SPL {X  -162.820, Y  +512.406, Z    +0.000, E1   -25.425, E3 +474181.954}
SPL {X  -162.820, Y  +515.039, Z    +0.000, E1   -25.452, E3 +474193.365}
SPL {X  -162.820, Y  +518.350, Z    +0.000, E1   -25.425, E3 +474208.114}
SPL {X  -162.820, Y  +521.486, Z    +0.000, E1   -25.382, E3 +474222.142}
SPL {X  -162.820, Y  +524.180, Z    +0.000, E1   -25.495, E3 +474233.014}
SPL {X  -162.820, Y  +527.020, Z    +0.000, E1   -25.477, E3 +474245.707}
SPL {X  -162.820, Y  +529.670, Z    +0.000, E1   -25.472, E3 +474257.165}
SPL {X  -162.820, Y  +532.006, Z    +0.000, E1   -25.455, E3 +474267.622}
SPL {X  -162.820, Y  +534.806, Z    +0.000, E1   -25.465, E3 +474279.738}
SPL {X  -162.820, Y  +537.226, Z    +0.000, E1   -25.378, E3 +474291.020}
SPL {X  -162.820, Y  +540.345, Z    +0.000, E1   -25.451, E3 +474304.201}
SPL {X  -162.820, Y  +543.279, Z    +0.000, E1   -25.419, E3 +474317.234}
SPL {X  -162.820, Y  +546.125, Z    +0.000, E1   -25.505, E3 +474329.028}
SPL {X  -162.820, Y  +549.578, Z    +0.000, E1   -25.462, E3 +474344.652}
SPL {X  -162.820, Y  +553.157, Z    +0.000, E1   -25.443, E3 +474360.316}
SPL {X  -162.820, Y  +556.150, Z    +0.000, E1   -25.445, E3 +474373.405}
SPL {X  -162.820, Y  +559.215, Z    +0.000, E1   -25.460, E3 +474386.707}
SPL {X  -162.820, Y  +562.125, Z    +0.000, E1   -25.434, E3 +474399.627}
SPL {X  -162.820, Y  +564.880, Z    +0.000, E1   -25.448, E3 +474411.581}
SPL {X  -162.820, Y  +568.326, Z    +0.000, E1   -25.470, E3 +474426.641}
SPL {X  -162.820, Y  +571.303, Z    +0.000, E1   -25.427, E3 +474439.814}
SPL {X  -162.820, Y  +574.067, Z    +0.000, E1   -25.459, E3 +474451.753}
SPL {X  -162.820, Y  +576.597, Z    +0.000, E1   -25.400, E3 +474463.224}
SPL {X  -162.820, Y  +578.977, Z    +0.000, E1   -25.460, E3 +474473.157}
SPL {X  -162.820, Y  +581.995, Z    +0.000, E1   -25.468, E3 +474486.515}
SPL {X  -162.820, Y  +585.512, Z    +0.000, E1   -25.448, E3 +474501.938}
SPL {X  -162.820, Y  +588.371, Z    +0.000, E1   -25.460, E3 +474514.324}
SPL {X  -162.820, Y  +591.246, Z    +0.000, E1   -25.415, E3 +474527.343}
SPL {X  -162.820, Y  +594.339, Z    +0.000, E1   -25.487, E3 +474540.246}
SPL {X  -162.820, Y  +596.868, Z    +0.000, E1   -25.461, E3 +474551.509}
SPL {X  -162.820, Y  +600.326, Z    +0.000, E1   -25.438, E3 +474567.030}
SPL {X  -162.820, Y  +604.526, Z    +0.000, E1   -25.502, E3 +474584.853}
SPL {X  -162.820, Y  +607.811, Z    +0.000, E1   -25.507, E3 +474599.068}
SPL {X  -162.820, Y  +610.517, Z    +0.000, E1   -25.412, E3 +474611.630}
SPL {X  -162.820, Y  +613.762, Z    +0.000, E1   -25.472, E3 +474625.437}
SPL {X  -162.820, Y  +617.275, Z    +0.000, E1   -25.466, E3 +474640.876}
SPL {X  -162.820, Y  +621.264, Z    +0.000, E1   -25.514, E3 +474658.037}
SPL {X  -162.820, Y  +624.430, Z    +0.000, E1   -25.475, E3 +474671.968}
SPL {X  -162.820, Y  +626.570, Z    +0.000, E1   -25.441, E3 +474681.569}
SPL {X  -162.820, Y  +628.902, Z    +0.000, E1   -25.449, E3 +474691.749}
SPL {X  -162.820, Y  +631.177, Z    +0.000, E1   -25.467, E3 +474701.580}
SPL {X  -162.820, Y  +633.994, Z    +0.000, E1   -25.503, E3 +474713.627}
SPL {X  -162.820, Y  +636.469, Z    +0.000, E1   -25.465, E3 +474724.670}
SPL {X  -162.820, Y  +638.486, Z    +0.000, E1   -25.456, E3 +474733.588}
SPL {X  -162.820, Y  +640.803, Z    +0.000, E1   -25.462, E3 +474743.649}
SPL {X  -162.820, Y  +643.028, Z    +0.000, E1   -25.494, E3 +474753.159}
SPL {X  -162.820, Y  +645.694, Z    +0.000, E1   -25.540, E3 +474764.446}
SPL {X  -162.820, Y  +649.102, Z    +0.000, E1   -25.495, E3 +474779.875}
SPL {X  -162.820, Y  +652.810, Z    +0.000, E1   -25.497, E3 +474795.908}
SPL {X  -162.820, Y  +655.214, Z    +0.000, E1   -25.485, E3 +474806.411}
SPL {X  -162.820, Y  +657.616, Z    +0.000, E1   -25.511, E3 +474816.765}
SPL {X  -162.820, Y  +660.851, Z    +0.000, E1   -25.520, E3 +474830.908}
SPL {X  -162.820, Y  +663.853, Z    +0.000, E1   -25.496, E3 +474844.089}
SPL {X  -162.820, Y  +666.096, Z    +0.000, E1   -25.408, E3 +474854.556}
SPL {X  -162.820, Y  +669.195, Z    +0.000, E1   -25.525, E3 +474867.393}
SPL {X  -162.820, Y  +672.979, Z    +0.000, E1   -25.478, E3 +474884.243}
SPL {X  -162.796, Y  +676.319, Z    +0.000, E1   -25.526, E3 +474898.388}
SPL {X  -162.739, Y  +678.625, Z    +0.000, E1   -25.423, E3 +474909.180}
SPL {X  -162.669, Y  +680.515, Z    +0.000, E1   -25.398, E3 +474917.634}
SPL {X  -162.545, Y  +682.952, Z    +0.000, E1   -25.510, E3 +474927.496}
SPL {X  -162.381, Y  +685.455, Z    +0.000, E1   -25.410, E3 +474939.182}
SPL {X  -162.194, Y  +687.760, Z    +0.000, E1   -25.360, E3 +474949.618}
SPL {X  -161.866, Y  +691.104, Z    +0.000, E1   -25.383, E3 +474964.250}
SPL {X  -161.024, Y  +697.619, Z    +0.000, E1   -26.780, E3 +474981.481}
SPL {X  -157.189, Y  +715.948, Z    +0.000, E1   -34.218, E3 +474996.400}
ENDSPLINE

SPLINE
SPL {X  -157.848, Y  +713.428, Z    +0.000, E1   -28.857, E3 +475030.539}
SPL {X  -161.035, Y  +697.541, Z    +0.000, E1   -20.899, E3 +475031.058}
SPL {X  -161.689, Y  +692.657, Z    +0.000, E1   -15.656, E3 +475071.141}
SPL {X  -162.807, Y  +675.545, Z    +0.000, E1    -5.787, E3 +475066.641}
ENDSPLINE

SPLINE
SPL {X  -162.791, Y  +676.574, Z    +0.000, E1    -6.127, E3 +475079.743}
ENDSPLINE

SPLINE
SPL {X  -162.820, Y  +664.716, Z    +0.000, E1    +1.705, E3 +475068.617}
SPL {X  -162.820, Y  +658.484, Z    +0.000, E1    +6.336, E3 +475075.094}
SPL {X  -162.820, Y  +640.102, Z    +0.000, E1   +22.409, E3 +475069.832}
SPL {X  -162.820, Y  +633.503, Z    +0.000, E1   +21.975, E3 +475102.069}
SPL {X  -162.820, Y  +611.299, Z    +0.000, E1   +31.088, E3 +475130.182}
ENDSPLINE

SPLINE
SPL {X  -162.820, Y  +618.877, Z    +0.000, E1   +25.259, E3 +475141.676}
ENDSPLINE

SPLINE
SPL {X  -162.820, Y  +617.582, Z    +0.000, E1   +24.552, E3 +475153.053}
SPL {X  -162.820, Y  +614.716, Z    +0.000, E1   +24.535, E3 +475166.264}
SPL {X  -162.820, Y  +611.754, Z    +0.000, E1   +24.563, E3 +475179.552}
SPL {X  -162.820, Y  +608.970, Z    +0.000, E1   +24.542, E3 +475192.393}
SPL {X  -162.820, Y  +606.285, Z    +0.000, E1   +24.533, E3 +475204.728}
SPL {X  -162.820, Y  +603.509, Z    +0.000, E1   +24.546, E3 +475217.265}
SPL {X  -162.820, Y  +600.818, Z    +0.000, E1   +24.590, E3 +475229.188}
SPL {X  -162.820, Y  +598.053, Z    +0.000, E1   +24.547, E3 +475242.171}
SPL {X  -162.820, Y  +595.188, Z    +0.000, E1   +24.538, E3 +475255.260}
SPL {X  -162.820, Y  +591.955, Z    +0.000, E1   +24.571, E3 +475269.880}
SPL {X  -162.820, Y  +587.913, Z    +0.000, E1   +24.604, E3 +475288.097}
SPL {X  -162.820, Y  +584.766, Z    +0.000, E1   +24.499, E3 +475303.077}
SPL {X  -162.820, Y  +581.896, Z    +0.000, E1   +24.528, E3 +475316.019}
SPL {X  -162.820, Y  +579.244, Z    +0.000, E1   +24.610, E3 +475327.363}
SPL {X  -162.820, Y  +576.848, Z    +0.000, E1   +24.543, E3 +475338.904}
SPL {X  -162.820, Y  +573.694, Z    +0.000, E1   +24.535, E3 +475353.374}
SPL {X  -162.820, Y  +571.322, Z    +0.000, E1   +24.492, E3 +475364.408}
SPL {X  -162.820, Y  +568.309, Z    +0.000, E1   +24.589, E3 +475377.633}
SPL {X  -162.820, Y  +564.977, Z    +0.000, E1   +24.571, E3 +475392.806}
SPL {X  -162.820, Y  +562.356, Z    +0.000, E1   +24.575, E3 +475404.704}
SPL {X  -162.820, Y  +558.990, Z    +0.000, E1   +24.558, E3 +475420.354}
SPL {X  -162.820, Y  +555.584, Z    +0.000, E1   +24.559, E3 +475435.723}
SPL {X  -162.820, Y  +552.867, Z    +0.000, E1   +24.583, E3 +475447.919}
SPL {X  -162.820, Y  +549.589, Z    +0.000, E1   +24.547, E3 +475463.285}
SPL {X  -162.820, Y  +546.972, Z    +0.000, E1   +24.516, E3 +475475.250}
SPL {X  -162.820, Y  +544.025, Z    +0.000, E1   +24.611, E3 +475488.194}
SPL {X  -162.820, Y  +540.573, Z    +0.000, E1   +24.503, E3 +475504.648}
SPL {X  -162.820, Y  +538.106, Z    +0.000, E1   +24.553, E3 +475515.402}
SPL {X  -162.820, Y  +536.451, Z    +0.000, E1   +24.519, E3 +475523.220}
SPL {X  -162.820, Y  +534.025, Z    +0.000, E1   +24.589, E3 +475533.821}
SPL {X  -162.820, Y  +531.527, Z    +0.000, E1   +24.582, E3 +475545.206}
SPL {X  -162.820, Y  +529.165, Z    +0.000, E1   +24.521, E3 +475556.455}
SPL {X  -162.820, Y  +525.802, Z    +0.000, E1   +24.585, E3 +475571.475}
SPL {X  -162.820, Y  +521.731, Z    +0.000, E1   +24.542, E3 +475590.411}
SPL {X  -162.820, Y  +518.185, Z    +0.000, E1   +24.561, E3 +475606.283}
SPL {X  -162.820, Y  +508.728, Z    +0.000, E1   +28.484, E3 +475616.823}
SPL {X  -162.820, Y  +500.664, Z    +0.000, E1   +31.476, E3 +475625.487}
SPL {X  -162.820, Y  +499.290, Z    +0.000, E1   +30.657, E3 +475635.769}
SPL {X  -162.820, Y  +497.700, Z    +0.000, E1   +29.785, E3 +475647.384}
SPL {X  -162.820, Y  +495.915, Z    +0.000, E1   +28.861, E3 +475660.476}
SPL {X  -162.820, Y  +494.678, Z    +0.000, E1   +27.647, E3 +475673.822}
SPL {X  -162.820, Y  +493.757, Z    +0.000, E1   +26.462, E3 +475686.182}
SPL {X  -162.820, Y  +491.420, Z    +0.000, E1   +25.780, E3 +475701.444}
SPL {X  -162.820, Y  +487.351, Z    +0.000, E1   +25.663, E3 +475719.960}
SPL {X  -162.820, Y  +484.247, Z    +0.000, E1   +25.651, E3 +475733.286}
SPL {X  -162.820, Y  +482.092, Z    +0.000, E1   +25.593, E3 +475743.113}
SPL {X  -162.820, Y  +479.578, Z    +0.000, E1   +25.634, E3 +475753.756}
SPL {X  -162.820, Y  +477.137, Z    +0.000, E1   +25.632, E3 +475764.335}
SPL {X  -162.820, Y  +473.770, Z    +0.000, E1   +25.664, E3 +475778.881}
SPL {X  -162.820, Y  +470.744, Z    +0.000, E1   +25.641, E3 +475791.978}
SPL {X  -162.820, Y  +467.745, Z    +0.000, E1   +25.668, E3 +475804.960}
SPL {X  -162.820, Y  +463.978, Z    +0.000, E1   +25.651, E3 +475821.437}
SPL {X  -162.820, Y  +459.882, Z    +0.000, E1   +25.674, E3 +475839.072}
SPL {X  -162.820, Y  +456.773, Z    +0.000, E1   +25.591, E3 +475853.018}
SPL {X  -162.820, Y  +453.678, Z    +0.000, E1   +25.652, E3 +475866.093}
SPL {X  -162.820, Y  +450.466, Z    +0.000, E1   +25.644, E3 +475880.038}
SPL {X  -162.820, Y  +447.822, Z    +0.000, E1   +25.664, E3 +475891.296}
SPL {X  -162.820, Y  +444.499, Z    +0.000, E1   +25.673, E3 +475905.867}
SPL {X  -162.820, Y  +440.857, Z    +0.000, E1   +25.614, E3 +475921.975}
SPL {X  -162.820, Y  +438.582, Z    +0.000, E1   +25.544, E3 +475932.295}
SPL {X  -162.820, Y  +435.635, Z    +0.000, E1   +25.661, E3 +475944.390}
SPL {X  -162.820, Y  +431.823, Z    +0.000, E1   +25.651, E3 +475961.039}
SPL {X  -162.820, Y  +428.576, Z    +0.000, E1   +25.647, E3 +475975.025}
SPL {X  -162.820, Y  +425.120, Z    +0.000, E1   +25.647, E3 +475990.209}
SPL {X  -162.820, Y  +420.840, Z    +0.000, E1   +25.658, E3 +476008.716}
SPL {X  -162.820, Y  +416.590, Z    +0.000, E1   +25.659, E3 +476027.160}
SPL {X  -162.820, Y  +412.302, Z    +0.000, E1   +25.662, E3 +476045.765}
SPL {X  -162.820, Y  +408.133, Z    +0.000, E1   +25.637, E3 +476064.023}
SPL {X  -162.820, Y  +404.293, Z    +0.000, E1   +25.628, E3 +476080.746}
SPL {X  -162.820, Y  +400.835, Z    +0.000, E1   +25.694, E3 +476095.146}
SPL {X  -162.820, Y  +398.703, Z    +0.000, E1   +25.586, E3 +476105.138}
SPL {X  -162.820, Y  +395.582, Z    +0.000, E1   +25.684, E3 +476118.129}
SPL {X  -162.820, Y  +391.417, Z    +0.000, E1   +25.659, E3 +476136.467}
SPL {X  -162.820, Y  +387.939, Z    +0.000, E1   +25.627, E3 +476151.614}
SPL {X  -162.820, Y  +385.565, Z    +0.000, E1   +25.686, E3 +476161.403}
SPL {X  -162.820, Y  +383.458, Z    +0.000, E1   +25.657, E3 +476170.767}
SPL {X  -162.820, Y  +380.448, Z    +0.000, E1   +25.674, E3 +476183.875}
SPL {X  -162.785, Y  +377.106, Z    +0.000, E1   +25.598, E3 +476198.820}
SPL {X  -162.709, Y  +374.484, Z    +0.000, E1   +25.711, E3 +476209.271}
SPL {X  -162.623, Y  +372.485, Z    +0.000, E1   +25.631, E3 +476218.551}
SPL {X  -162.487, Y  +370.088, Z    +0.000, E1   +25.525, E3 +476229.805}
SPL {X  -162.243, Y  +366.801, Z    +0.000, E1   +25.618, E3 +476243.445}
SPL {X  -161.977, Y  +363.953, Z    +0.000, E1   +25.528, E3 +476256.372}
SPL {X  -161.695, Y  +361.389, Z    +0.000, E1   +25.445, E3 +476268.187}
SPL {X  -161.190, Y  +357.520, Z    +0.000, E1   +25.774, E3 +476282.439}
SPL {X  -155.035, Y  +330.756, Z    +0.000, E1   +37.918, E3 +476292.940}
SPL {X  -153.918, Y  +327.401, Z    +0.000, E1   +34.677, E3 +476328.240}
ENDSPLINE

SPLINE
SPL {X  -159.701, Y  +348.785, Z    +0.000, E1   +24.361, E3 +476335.721}
SPL {X  -161.904, Y  +363.251, Z    +0.000, E1   +14.606, E3 +476365.516}
SPL {X  -162.745, Y  +375.561, Z    +0.000, E1    +7.538, E3 +476365.713}
SPL {X  -162.820, Y  +385.424, Z    +0.000, E1    +1.080, E3 +476366.607}
SPL {X  -162.820, Y  +389.940, Z    +0.000, E1    -2.281, E3 +476369.484}
SPL {X  -162.820, Y  +396.652, Z    +0.000, E1    -7.520, E3 +476369.062}
SPL {X  -162.820, Y  +406.605, Z    +0.000, E1   -16.760, E3 +476361.539}
SPL {X  -162.820, Y  +418.675, Z    +0.000, E1   -22.201, E3 +476387.788}
SPL {X  -162.820, Y  +425.113, Z    +0.000, E1   -25.243, E3 +476396.724}
SPL {X  -162.820, Y  +441.937, Z    +0.000, E1   -31.578, E3 +476418.802}
ENDSPLINE

SPLINE
SPL {X  -162.820, Y  +437.771, Z    +0.000, E1   -26.555, E3 +476437.903}
ENDSPLINE

SPLINE
SPL {X  -162.820, Y  +439.120, Z    +0.000, E1   -25.352, E3 +476452.446}
SPL {X  -162.820, Y  +441.593, Z    +0.000, E1   -25.391, E3 +476462.998}
SPL {X  -162.820, Y  +444.317, Z    +0.000, E1   -25.492, E3 +476474.179}
SPL {X  -162.820, Y  +446.544, Z    +0.000, E1   -25.427, E3 +476484.349}
SPL {X  -162.820, Y  +448.500, Z    +0.000, E1   -25.425, E3 +476492.950}
SPL {X  -162.820, Y  +451.056, Z    +0.000, E1   -25.443, E3 +476504.057}
SPL {X  -162.820, Y  +454.662, Z    +0.000, E1   -25.474, E3 +476519.802}
SPL {X  -162.820, Y  +458.079, Z    +0.000, E1   -25.369, E3 +476535.381}
SPL {X  -162.820, Y  +460.719, Z    +0.000, E1   -25.411, E3 +476546.639}
SPL {X  -162.820, Y  +463.419, Z    +0.000, E1   -25.510, E3 +476557.677}
SPL {X  -162.820, Y  +465.376, Z    +0.000, E1   -25.372, E3 +476567.264}
SPL {X  -162.820, Y  +467.440, Z    +0.000, E1   -25.427, E3 +476575.896}
SPL {X  -162.820, Y  +470.010, Z    +0.000, E1   -25.445, E3 +476587.101}
SPL {X  -162.820, Y  +473.445, Z    +0.000, E1   -25.493, E3 +476601.824}
SPL {X  -162.820, Y  +476.157, Z    +0.000, E1   -25.426, E3 +476614.039}
SPL {X  -162.820, Y  +478.461, Z    +0.000, E1   -25.410, E3 +476624.319}
SPL {X  -162.820, Y  +480.780, Z    +0.000, E1   -25.447, E3 +476634.181}
SPL {X  -162.820, Y  +483.622, Z    +0.000, E1   -25.381, E3 +476647.223}
SPL {X  -162.820, Y  +487.570, Z    +0.000, E1   -25.482, E3 +476663.861}
SPL {X  -162.820, Y  +491.017, Z    +0.000, E1   -25.445, E3 +476679.075}
SPL {X  -162.820, Y  +493.705, Z    +0.000, E1   -25.443, E3 +476690.860}
SPL {X  -162.820, Y  +497.247, Z    +0.000, E1   -25.470, E3 +476706.322}
SPL {X  -162.820, Y  +501.343, Z    +0.000, E1   -25.435, E3 +476724.521}
SPL {X  -162.820, Y  +505.370, Z    +0.000, E1   -25.456, E3 +476741.984}
SPL {X  -162.820, Y  +509.412, Z    +0.000, E1   -25.458, E3 +476759.707}
SPL {X  -162.820, Y  +512.406, Z    +0.000, E1   -25.425, E3 +476772.863}
SPL {X  -162.820, Y  +515.039, Z    +0.000, E1   -25.452, E3 +476784.274}
SPL {X  -162.820, Y  +518.350, Z    +0.000, E1   -25.425, E3 +476799.023}
SPL {X  -162.820, Y  +521.486, Z    +0.000, E1   -25.382, E3 +476813.051}
SPL {X  -162.820, Y  +524.180, Z    +0.000, E1   -25.495, E3 +476823.923}
SPL {X  -162.820, Y  +527.020, Z    +0.000, E1   -25.477, E3 +476836.616}
SPL {X  -162.820, Y  +529.670, Z    +0.000, E1   -25.472, E3 +476848.074}
SPL {X  -162.820, Y  +532.006, Z    +0.000, E1   -25.455, E3 +476858.531}
SPL {X  -162.820, Y  +534.806, Z    +0.000, E1   -25.465, E3 +476870.647}
SPL {X  -162.820, Y  +537.226, Z    +0.000, E1   -25.378, E3 +476881.929}
SPL {X  -162.820, Y  +539.521, Z    +0.000, E1   -25.386, E3 +476891.887}
SPL {X  -162.820, Y  +542.667, Z    +0.000, E1   -25.474, E3 +476905.212}
SPL {X  -162.820, Y  +546.125, Z    +0.000, E1   -25.505, E3 +476919.937}
SPL {X  -162.820, Y  +548.232, Z    +0.000, E1   -25.424, E3 +476929.699}
SPL {X  -162.820, Y  +550.399, Z    +0.000, E1   -25.424, E3 +476939.251}
SPL {X  -162.820, Y  +553.157, Z    +0.000, E1   -25.443, E3 +476951.225}
SPL {X  -162.820, Y  +556.965, Z    +0.000, E1   -25.478, E3 +476967.817}
SPL {X  -162.820, Y  +561.429, Z    +0.000, E1   -25.478, E3 +476987.336}
SPL {X  -162.820, Y  +565.606, Z    +0.000, E1   -25.468, E3 +477005.666}
SPL {X  -162.820, Y  +568.974, Z    +0.000, E1   -25.453, E3 +477020.376}
SPL {X  -162.820, Y  +571.303, Z    +0.000, E1   -25.427, E3 +477030.723}
SPL {X  -162.820, Y  +574.067, Z    +0.000, E1   -25.459, E3 +477042.662}
SPL {X  -162.820, Y  +576.597, Z    +0.000, E1   -25.400, E3 +477054.133}
SPL {X  -162.820, Y  +578.977, Z    +0.000, E1   -25.460, E3 +477064.066}
SPL {X  -162.820, Y  +581.995, Z    +0.000, E1   -25.468, E3 +477077.424}
SPL {X  -162.820, Y  +585.512, Z    +0.000, E1   -25.448, E3 +477092.847}
SPL {X  -162.820, Y  +588.371, Z    +0.000, E1   -25.460, E3 +477105.233}
SPL {X  -162.820, Y  +591.246, Z    +0.000, E1   -25.415, E3 +477118.252}
SPL {X  -162.820, Y  +594.339, Z    +0.000, E1   -25.487, E3 +477131.155}
SPL {X  -162.820, Y  +596.868, Z    +0.000, E1   -25.461, E3 +477142.418}
SPL {X  -162.820, Y  +600.326, Z    +0.000, E1   -25.438, E3 +477157.939}
SPL {X  -162.820, Y  +604.526, Z    +0.000, E1   -25.502, E3 +477175.762}
SPL {X  -162.820, Y  +607.811, Z    +0.000, E1   -25.507, E3 +477189.977}
SPL {X  -162.820, Y  +610.517, Z    +0.000, E1   -25.412, E3 +477202.539}
SPL {X  -162.820, Y  +613.762, Z    +0.000, E1   -25.472, E3 +477216.346}
SPL {X  -162.820, Y  +617.275, Z    +0.000, E1   -25.466, E3 +477231.785}
SPL {X  -162.820, Y  +621.264, Z    +0.000, E1   -25.514, E3 +477248.947}
SPL {X  -162.820, Y  +624.430, Z    +0.000, E1   -25.475, E3 +477262.877}
SPL {X  -162.820, Y  +626.570, Z    +0.000, E1   -25.441, E3 +477272.478}
SPL {X  -162.820, Y  +628.902, Z    +0.000, E1   -25.449, E3 +477282.658}
SPL {X  -162.820, Y  +631.177, Z    +0.000, E1   -25.467, E3 +477292.489}
SPL {X  -162.820, Y  +633.994, Z    +0.000, E1   -25.503, E3 +477304.536}
SPL {X  -162.820, Y  +636.469, Z    +0.000, E1   -25.465, E3 +477315.579}
SPL {X  -162.820, Y  +638.486, Z    +0.000, E1   -25.456, E3 +477324.497}
SPL {X  -162.820, Y  +640.803, Z    +0.000, E1   -25.462, E3 +477334.559}
SPL {X  -162.820, Y  +643.028, Z    +0.000, E1   -25.494, E3 +477344.068}
SPL {X  -162.820, Y  +645.694, Z    +0.000, E1   -25.540, E3 +477355.356}
SPL {X  -162.820, Y  +649.102, Z    +0.000, E1   -25.495, E3 +477370.784}
SPL {X  -162.820, Y  +652.810, Z    +0.000, E1   -25.497, E3 +477386.817}
SPL {X  -162.820, Y  +655.214, Z    +0.000, E1   -25.485, E3 +477397.320}
SPL {X  -162.820, Y  +657.616, Z    +0.000, E1   -25.511, E3 +477407.674}
SPL {X  -162.820, Y  +660.007, Z    +0.000, E1   -25.550, E3 +477417.736}
SPL {X  -162.820, Y  +662.980, Z    +0.000, E1   -25.505, E3 +477431.294}
SPL {X  -162.820, Y  +667.253, Z    +0.000, E1   -25.483, E3 +477450.171}
SPL {X  -162.820, Y  +671.102, Z    +0.000, E1   -25.514, E3 +477466.621}
SPL {X  -162.820, Y  +673.648, Z    +0.000, E1   -25.431, E3 +477478.288}
SPL {X  -162.796, Y  +676.319, Z    +0.000, E1   -25.526, E3 +477489.297}
SPL {X  -162.707, Y  +679.552, Z    +0.000, E1   -25.443, E3 +477504.172}
SPL {X  -162.545, Y  +682.952, Z    +0.000, E1   -25.510, E3 +477518.405}
SPL {X  -162.381, Y  +685.455, Z    +0.000, E1   -25.410, E3 +477530.092}
SPL {X  -162.102, Y  +688.774, Z    +0.000, E1   -25.417, E3 +477544.706}
SPL {X  -161.778, Y  +691.887, Z    +0.000, E1   -25.301, E3 +477559.007}
SPL {X  -161.319, Y  +695.558, Z    +0.000, E1   -25.832, E3 +477570.962}
SPL {X  -157.976, Y  +712.921, Z    +0.000, E1   -33.197, E3 +477584.353}
ENDSPLINE

SPLINE
SPL {X  -160.738, Y  +699.453, Z    +0.000, E1   -21.994, E3 +477621.980}
SPL {X  -161.689, Y  +692.657, Z    +0.000, E1   -15.656, E3 +477662.050}
SPL {X  -162.807, Y  +675.545, Z    +0.000, E1    -5.787, E3 +477657.550}
ENDSPLINE

SPLINE
SPL {X  -162.791, Y  +676.574, Z    +0.000, E1    -6.127, E3 +477670.652}
ENDSPLINE

SPLINE
SPL {X  -162.820, Y  +664.716, Z    +0.000, E1    +1.705, E3 +477659.527}
SPL {X  -162.820, Y  +658.484, Z    +0.000, E1    +6.336, E3 +477666.003}
SPL {X  -162.820, Y  +640.102, Z    +0.000, E1   +22.409, E3 +477660.742}
SPL {X  -162.820, Y  +633.503, Z    +0.000, E1   +21.975, E3 +477692.978}
SPL {X  -162.820, Y  +611.299, Z    +0.000, E1   +31.088, E3 +477721.091}
ENDSPLINE

SPLINE
SPL {X  -162.820, Y  +618.877, Z    +0.000, E1   +25.259, E3 +477732.585}
ENDSPLINE

SPLINE
SPL {X  -162.820, Y  +617.582, Z    +0.000, E1   +24.552, E3 +477743.962}
SPL {X  -162.820, Y  +614.716, Z    +0.000, E1   +24.535, E3 +477757.173}
SPL {X  -162.820, Y  +611.754, Z    +0.000, E1   +24.563, E3 +477770.461}
SPL {X  -162.820, Y  +608.970, Z    +0.000, E1   +24.542, E3 +477783.302}
SPL {X  -162.820, Y  +606.285, Z    +0.000, E1   +24.533, E3 +477795.637}
SPL {X  -162.820, Y  +603.509, Z    +0.000, E1   +24.546, E3 +477808.174}
SPL {X  -162.820, Y  +600.818, Z    +0.000, E1   +24.590, E3 +477820.097}
SPL {X  -162.820, Y  +598.053, Z    +0.000, E1   +24.547, E3 +477833.080}
SPL {X  -162.820, Y  +595.188, Z    +0.000, E1   +24.538, E3 +477846.169}
SPL {X  -162.820, Y  +592.738, Z    +0.000, E1   +24.551, E3 +477857.217}
SPL {X  -162.820, Y  +590.118, Z    +0.000, E1   +24.544, E3 +477869.276}
SPL {X  -162.820, Y  +587.204, Z    +0.000, E1   +24.592, E3 +477882.153}
SPL {X  -162.820, Y  +584.193, Z    +0.000, E1   +24.484, E3 +477896.863}
SPL {X  -162.820, Y  +580.163, Z    +0.000, E1   +24.634, E3 +477914.098}
SPL {X  -162.820, Y  +576.848, Z    +0.000, E1   +24.543, E3 +477929.814}
SPL {X  -162.820, Y  +574.433, Z    +0.000, E1   +24.551, E3 +477940.644}
SPL {X  -162.820, Y  +572.074, Z    +0.000, E1   +24.505, E3 +477951.915}
SPL {X  -162.820, Y  +569.438, Z    +0.000, E1   +24.562, E3 +477963.374}
SPL {X  -162.820, Y  +567.494, Z    +0.000, E1   +24.547, E3 +477972.385}
SPL {X  -162.820, Y  +564.977, Z    +0.000, E1   +24.571, E3 +477983.715}
SPL {X  -162.820, Y  +562.356, Z    +0.000, E1   +24.575, E3 +477995.613}
SPL {X  -162.820, Y  +560.119, Z    +0.000, E1   +24.506, E3 +478006.302}
SPL {X  -162.820, Y  +558.093, Z    +0.000, E1   +24.537, E3 +478015.320}
SPL {X  -162.820, Y  +555.584, Z    +0.000, E1   +24.559, E3 +478026.632}
SPL {X  -162.820, Y  +552.169, Z    +0.000, E1   +24.581, E3 +478042.201}
SPL {X  -162.820, Y  +548.932, Z    +0.000, E1   +24.540, E3 +478057.102}
SPL {X  -162.820, Y  +545.742, Z    +0.000, E1   +24.577, E3 +478071.481}
SPL {X  -162.820, Y  +542.142, Z    +0.000, E1   +24.582, E3 +478087.834}
SPL {X  -162.820, Y  +538.903, Z    +0.000, E1   +24.519, E3 +478103.050}
SPL {X  -162.820, Y  +536.451, Z    +0.000, E1   +24.519, E3 +478114.130}
SPL {X  -162.820, Y  +534.025, Z    +0.000, E1   +24.589, E3 +478124.730}
SPL {X  -162.820, Y  +531.527, Z    +0.000, E1   +24.582, E3 +478136.115}
SPL {X  -162.820, Y  +529.165, Z    +0.000, E1   +24.521, E3 +478147.364}
SPL {X  -162.820, Y  +526.822, Z    +0.000, E1   +24.559, E3 +478157.727}
SPL {X  -162.820, Y  +524.112, Z    +0.000, E1   +24.542, E3 +478170.345}
SPL {X  -162.820, Y  +521.048, Z    +0.000, E1   +24.515, E3 +478184.481}
SPL {X  -162.820, Y  +518.185, Z    +0.000, E1   +24.561, E3 +478197.192}
SPL {X  -162.820, Y  +508.728, Z    +0.000, E1   +28.484, E3 +478207.732}
SPL {X  -162.820, Y  +500.664, Z    +0.000, E1   +31.476, E3 +478216.396}
SPL {X  -162.820, Y  +499.290, Z    +0.000, E1   +30.657, E3 +478226.678}
SPL {X  -162.820, Y  +497.251, Z    +0.000, E1   +29.634, E3 +478241.154}
SPL {X  -162.820, Y  +495.647, Z    +0.000, E1   +28.606, E3 +478254.030}
SPL {X  -162.820, Y  +494.678, Z    +0.000, E1   +27.647, E3 +478264.731}
SPL {X  -162.820, Y  +493.757, Z    +0.000, E1   +26.462, E3 +478277.091}
SPL {X  -162.820, Y  +492.330, Z    +0.000, E1   +25.953, E3 +478286.845}
SPL {X  -162.820, Y  +489.800, Z    +0.000, E1   +25.653, E3 +478300.307}
SPL {X  -162.820, Y  +485.392, Z    +0.000, E1   +25.667, E3 +478319.334}
SPL {X  -162.820, Y  +482.092, Z    +0.000, E1   +25.593, E3 +478334.022}
SPL {X  -162.820, Y  +479.578, Z    +0.000, E1   +25.634, E3 +478344.665}
SPL {X  -162.820, Y  +477.137, Z    +0.000, E1   +25.632, E3 +478355.244}
SPL {X  -162.820, Y  +473.770, Z    +0.000, E1   +25.664, E3 +478369.790}
SPL {X  -162.820, Y  +469.694, Z    +0.000, E1   +25.657, E3 +478387.521}
SPL {X  -162.820, Y  +465.727, Z    +0.000, E1   +25.676, E3 +478404.564}
SPL {X  -162.820, Y  +463.001, Z    +0.000, E1   +25.614, E3 +478416.680}
SPL {X  -162.820, Y  +459.882, Z    +0.000, E1   +25.674, E3 +478429.981}
SPL {X  -162.820, Y  +456.773, Z    +0.000, E1   +25.591, E3 +478443.927}
SPL {X  -162.820, Y  +454.429, Z    +0.000, E1   +25.642, E3 +478453.695}
SPL {X  -162.820, Y  +451.204, Z    +0.000, E1   +25.672, E3 +478467.722}
SPL {X  -162.820, Y  +447.822, Z    +0.000, E1   +25.664, E3 +478482.205}
SPL {X  -162.820, Y  +445.556, Z    +0.000, E1   +25.626, E3 +478492.336}
SPL {X  -162.820, Y  +442.508, Z    +0.000, E1   +25.657, E3 +478505.430}
SPL {X  -162.820, Y  +439.273, Z    +0.000, E1   +25.576, E3 +478520.068}
SPL {X  -162.820, Y  +436.773, Z    +0.000, E1   +25.602, E3 +478530.633}
SPL {X  -162.820, Y  +433.761, Z    +0.000, E1   +25.681, E3 +478543.311}
SPL {X  -162.820, Y  +430.942, Z    +0.000, E1   +25.597, E3 +478555.996}
SPL {X  -162.820, Y  +428.576, Z    +0.000, E1   +25.647, E3 +478565.934}
SPL {X  -162.820, Y  +426.525, Z    +0.000, E1   +25.610, E3 +478575.041}
SPL {X  -162.820, Y  +423.655, Z    +0.000, E1   +25.628, E3 +478587.601}
SPL {X  -162.820, Y  +419.407, Z    +0.000, E1   +25.665, E3 +478605.794}
SPL {X  -162.820, Y  +415.900, Z    +0.000, E1   +25.638, E3 +478621.063}
SPL {X  -162.820, Y  +413.088, Z    +0.000, E1   +25.644, E3 +478633.219}
SPL {X  -162.820, Y  +410.320, Z    +0.000, E1   +25.604, E3 +478645.538}
SPL {X  -162.820, Y  +407.487, Z    +0.000, E1   +25.617, E3 +478657.746}
SPL {X  -162.820, Y  +405.108, Z    +0.000, E1   +25.535, E3 +478668.713}
SPL {X  -162.820, Y  +401.373, Z    +0.000, E1   +25.736, E3 +478683.550}
SPL {X  -162.820, Y  +398.703, Z    +0.000, E1   +25.586, E3 +478696.047}
SPL {X  -162.820, Y  +395.582, Z    +0.000, E1   +25.684, E3 +478709.038}
SPL {X  -162.820, Y  +391.417, Z    +0.000, E1   +25.659, E3 +478727.376}
SPL {X  -162.820, Y  +387.939, Z    +0.000, E1   +25.627, E3 +478742.523}
SPL {X  -162.820, Y  +385.565, Z    +0.000, E1   +25.686, E3 +478752.312}
SPL {X  -162.820, Y  +383.458, Z    +0.000, E1   +25.657, E3 +478761.676}
SPL {X  -162.820, Y  +381.229, Z    +0.000, E1   +25.660, E3 +478771.351}
SPL {X  -162.797, Y  +377.786, Z    +0.000, E1   +25.638, E3 +478786.641}
SPL {X  -162.663, Y  +373.346, Z    +0.000, E1   +25.707, E3 +478805.380}
SPL {X  -162.487, Y  +370.088, Z    +0.000, E1   +25.525, E3 +478820.714}
SPL {X  -162.307, Y  +367.587, Z    +0.000, E1   +25.577, E3 +478831.133}
SPL {X  -162.041, Y  +364.588, Z    +0.000, E1   +25.591, E3 +478844.210}
SPL {X  -161.695, Y  +361.389, Z    +0.000, E1   +25.445, E3 +478859.096}
SPL {X  -161.190, Y  +357.520, Z    +0.000, E1   +25.774, E3 +478873.348}
SPL {X  -155.035, Y  +330.756, Z    +0.000, E1   +37.918, E3 +478883.849}
SPL {X  -153.918, Y  +327.401, Z    +0.000, E1   +34.677, E3 +478919.150}
ENDSPLINE

SPLINE
SPL {X  -159.701, Y  +348.785, Z    +0.000, E1   +24.361, E3 +478926.630}
SPL {X  -161.904, Y  +363.251, Z    +0.000, E1   +14.606, E3 +478956.425}
SPL {X  -162.745, Y  +375.561, Z    +0.000, E1    +7.538, E3 +478956.622}
SPL {X  -162.820, Y  +385.424, Z    +0.000, E1    +1.080, E3 +478957.516}
SPL {X  -162.820, Y  +389.940, Z    +0.000, E1    -2.281, E3 +478960.393}
SPL {X  -162.820, Y  +396.652, Z    +0.000, E1    -7.520, E3 +478959.971}
SPL {X  -162.820, Y  +406.605, Z    +0.000, E1   -16.760, E3 +478952.448}
SPL {X  -162.820, Y  +420.013, Z    +0.000, E1   -22.833, E3 +478980.569}
SPL {X  -162.820, Y  +442.075, Z    +0.000, E1   -31.090, E3 +479013.355}
ENDSPLINE

SPLINE
SPL {X  -162.820, Y  +436.680, Z    +0.000, E1   -26.151, E3 +479026.660}
ENDSPLINE

SPLINE
SPL {X  -162.820, Y  +438.487, Z    +0.000, E1   -25.409, E3 +479040.298}
SPL {X  -162.820, Y  +441.593, Z    +0.000, E1   -25.391, E3 +479053.907}
SPL {X  -162.820, Y  +444.317, Z    +0.000, E1   -25.492, E3 +479065.088}
SPL {X  -162.820, Y  +447.641, Z    +0.000, E1   -25.460, E3 +479080.023}
SPL {X  -162.820, Y  +451.939, Z    +0.000, E1   -25.468, E3 +479098.843}
SPL {X  -162.820, Y  +455.480, Z    +0.000, E1   -25.454, E3 +479114.255}
SPL {X  -162.820, Y  +458.079, Z    +0.000, E1   -25.369, E3 +479126.290}
SPL {X  -162.820, Y  +460.719, Z    +0.000, E1   -25.411, E3 +479137.548}
SPL {X  -162.820, Y  +463.419, Z    +0.000, E1   -25.510, E3 +479148.586}
SPL {X  -162.820, Y  +466.458, Z    +0.000, E1   -25.433, E3 +479162.642}
SPL {X  -162.820, Y  +470.010, Z    +0.000, E1   -25.445, E3 +479178.010}
SPL {X  -162.820, Y  +472.345, Z    +0.000, E1   -25.448, E3 +479188.097}
SPL {X  -162.820, Y  +475.191, Z    +0.000, E1   -25.489, E3 +479200.459}
SPL {X  -162.820, Y  +478.461, Z    +0.000, E1   -25.410, E3 +479215.228}
SPL {X  -162.820, Y  +480.780, Z    +0.000, E1   -25.447, E3 +479225.090}
SPL {X  -162.820, Y  +483.622, Z    +0.000, E1   -25.381, E3 +479238.132}
SPL {X  -162.820, Y  +487.570, Z    +0.000, E1   -25.482, E3 +479254.770}
SPL {X  -162.820, Y  +491.017, Z    +0.000, E1   -25.445, E3 +479269.984}
SPL {X  -162.820, Y  +493.705, Z    +0.000, E1   -25.443, E3 +479281.769}
SPL {X  -162.820, Y  +497.247, Z    +0.000, E1   -25.470, E3 +479297.231}
SPL {X  -162.820, Y  +501.343, Z    +0.000, E1   -25.435, E3 +479315.430}
SPL {X  -162.820, Y  +505.370, Z    +0.000, E1   -25.456, E3 +479332.894}
SPL {X  -162.820, Y  +509.412, Z    +0.000, E1   -25.458, E3 +479350.616}
SPL {X  -162.820, Y  +512.406, Z    +0.000, E1   -25.425, E3 +479363.772}
SPL {X  -162.820, Y  +515.039, Z    +0.000, E1   -25.452, E3 +479375.183}
SPL {X  -162.820, Y  +518.350, Z    +0.000, E1   -25.425, E3 +479389.932}
SPL {X  -162.820, Y  +521.486, Z    +0.000, E1   -25.382, E3 +479403.960}
SPL {X  -162.820, Y  +524.180, Z    +0.000, E1   -25.495, E3 +479414.832}
SPL {X  -162.820, Y  +527.020, Z    +0.000, E1   -25.477, E3 +479427.525}
SPL {X  -162.820, Y  +529.670, Z    +0.000, E1   -25.472, E3 +479438.983}
SPL {X  -162.820, Y  +532.006, Z    +0.000, E1   -25.455, E3 +479449.440}
SPL {X  -162.820, Y  +534.806, Z    +0.000, E1   -25.465, E3 +479461.556}
SPL {X  -162.820, Y  +537.226, Z    +0.000, E1   -25.378, E3 +479472.838}
SPL {X  -162.820, Y  +540.345, Z    +0.000, E1   -25.451, E3 +479486.019}
SPL {X  -162.820, Y  +543.279, Z    +0.000, E1   -25.419, E3 +479499.052}
SPL {X  -162.820, Y  +546.125, Z    +0.000, E1   -25.505, E3 +479510.846}
SPL {X  -162.820, Y  +549.578, Z    +0.000, E1   -25.462, E3 +479526.470}
SPL {X  -162.820, Y  +553.157, Z    +0.000, E1   -25.443, E3 +479542.134}
SPL {X  -162.820, Y  +556.150, Z    +0.000, E1   -25.445, E3 +479555.223}
SPL {X  -162.820, Y  +559.215, Z    +0.000, E1   -25.460, E3 +479568.525}
SPL {X  -162.820, Y  +562.125, Z    +0.000, E1   -25.434, E3 +479581.445}
SPL {X  -162.820, Y  +564.880, Z    +0.000, E1   -25.448, E3 +479593.400}
SPL {X  -162.820, Y  +568.326, Z    +0.000, E1   -25.470, E3 +479608.459}
SPL {X  -162.820, Y  +571.303, Z    +0.000, E1   -25.427, E3 +479621.632}
SPL {X  -162.820, Y  +574.067, Z    +0.000, E1   -25.459, E3 +479633.571}
SPL {X  -162.820, Y  +576.597, Z    +0.000, E1   -25.400, E3 +479645.042}
SPL {X  -162.820, Y  +578.977, Z    +0.000, E1   -25.460, E3 +479654.975}
SPL {X  -162.820, Y  +581.995, Z    +0.000, E1   -25.468, E3 +479668.333}
SPL {X  -162.820, Y  +585.512, Z    +0.000, E1   -25.448, E3 +479683.756}
SPL {X  -162.820, Y  +588.371, Z    +0.000, E1   -25.460, E3 +479696.142}
SPL {X  -162.820, Y  +591.246, Z    +0.000, E1   -25.415, E3 +479709.161}
SPL {X  -162.820, Y  +594.339, Z    +0.000, E1   -25.487, E3 +479722.064}
SPL {X  -162.820, Y  +596.868, Z    +0.000, E1   -25.461, E3 +479733.327}
SPL {X  -162.820, Y  +600.326, Z    +0.000, E1   -25.438, E3 +479748.848}
SPL {X  -162.820, Y  +604.526, Z    +0.000, E1   -25.502, E3 +479766.672}
SPL {X  -162.820, Y  +607.811, Z    +0.000, E1   -25.507, E3 +479780.886}
SPL {X  -162.820, Y  +610.517, Z    +0.000, E1   -25.412, E3 +479793.449}
SPL {X  -162.820, Y  +613.762, Z    +0.000, E1   -25.472, E3 +479807.255}
SPL {X  -162.820, Y  +616.216, Z    +0.000, E1   -25.419, E3 +479818.251}
SPL {X  -162.820, Y  +618.995, Z    +0.000, E1   -25.483, E3 +479830.101}
SPL {X  -162.820, Y  +622.118, Z    +0.000, E1   -25.492, E3 +479843.566}
SPL {X  -162.820, Y  +624.430, Z    +0.000, E1   -25.475, E3 +479853.787}
SPL {X  -162.820, Y  +626.570, Z    +0.000, E1   -25.441, E3 +479863.387}
SPL {X  -162.820, Y  +628.902, Z    +0.000, E1   -25.449, E3 +479873.567}
SPL {X  -162.820, Y  +631.177, Z    +0.000, E1   -25.467, E3 +479883.399}
SPL {X  -162.820, Y  +633.994, Z    +0.000, E1   -25.503, E3 +479895.445}
SPL {X  -162.820, Y  +636.469, Z    +0.000, E1   -25.465, E3 +479906.488}
SPL {X  -162.820, Y  +638.486, Z    +0.000, E1   -25.456, E3 +479915.406}
SPL {X  -162.820, Y  +640.803, Z    +0.000, E1   -25.462, E3 +479925.468}
SPL {X  -162.820, Y  +643.028, Z    +0.000, E1   -25.494, E3 +479934.977}
SPL {X  -162.820, Y  +645.694, Z    +0.000, E1   -25.540, E3 +479946.265}
SPL {X  -162.820, Y  +649.102, Z    +0.000, E1   -25.495, E3 +479961.693}
SPL {X  -162.820, Y  +652.810, Z    +0.000, E1   -25.497, E3 +479977.726}
SPL {X  -162.820, Y  +655.214, Z    +0.000, E1   -25.485, E3 +479988.229}
SPL {X  -162.820, Y  +657.616, Z    +0.000, E1   -25.511, E3 +479998.583}
SPL {X  -162.820, Y  +660.007, Z    +0.000, E1   -25.550, E3 +480008.645}
SPL {X  -162.820, Y  +662.980, Z    +0.000, E1   -25.505, E3 +480022.203}
SPL {X  -162.820, Y  +667.253, Z    +0.000, E1   -25.483, E3 +480041.080}
SPL {X  -162.820, Y  +671.102, Z    +0.000, E1   -25.514, E3 +480057.530}
SPL {X  -162.820, Y  +673.648, Z    +0.000, E1   -25.431, E3 +480069.197}
SPL {X  -162.796, Y  +676.319, Z    +0.000, E1   -25.526, E3 +480080.206}
SPL {X  -162.707, Y  +679.552, Z    +0.000, E1   -25.443, E3 +480095.081}
SPL {X  -162.545, Y  +682.952, Z    +0.000, E1   -25.510, E3 +480109.314}
SPL {X  -162.381, Y  +685.455, Z    +0.000, E1   -25.410, E3 +480121.001}
SPL {X  -162.102, Y  +688.774, Z    +0.000, E1   -25.417, E3 +480135.615}
SPL {X  -161.711, Y  +692.468, Z    +0.000, E1   -25.300, E3 +480152.588}
SPL {X  -161.141, Y  +696.825, Z    +0.000, E1   -26.170, E3 +480164.722}
SPL {X  -157.976, Y  +712.921, Z    +0.000, E1   -33.197, E3 +480175.262}
ENDSPLINE

SPLINE
SPL {X  -160.738, Y  +699.453, Z    +0.000, E1   -21.994, E3 +480212.889}
SPL {X  -161.689, Y  +692.657, Z    +0.000, E1   -15.656, E3 +480252.959}
SPL {X  -162.807, Y  +675.545, Z    +0.000, E1    -5.787, E3 +480248.459}
ENDSPLINE

SPLINE
SPL {X  -162.791, Y  +676.574, Z    +0.000, E1    -6.127, E3 +480261.562}
ENDSPLINE

SPLINE
SPL {X  -162.820, Y  +664.716, Z    +0.000, E1    +1.705, E3 +480250.436}
SPL {X  -162.820, Y  +658.484, Z    +0.000, E1    +6.336, E3 +480256.912}
SPL {X  -162.820, Y  +640.102, Z    +0.000, E1   +22.409, E3 +480251.651}
SPL {X  -162.820, Y  +633.503, Z    +0.000, E1   +21.975, E3 +480283.887}
SPL {X  -162.820, Y  +611.299, Z    +0.000, E1   +31.088, E3 +480312.000}
ENDSPLINE

SPLINE
SPL {X  -162.820, Y  +618.877, Z    +0.000, E1   +25.259, E3 +480323.494}
ENDSPLINE

SPLINE
SPL {X  -162.820, Y  +617.582, Z    +0.000, E1   +24.552, E3 +480334.871}
SPL {X  -162.820, Y  +614.716, Z    +0.000, E1   +24.535, E3 +480348.082}
SPL {X  -162.820, Y  +611.754, Z    +0.000, E1   +24.563, E3 +480361.370}
SPL {X  -162.820, Y  +608.970, Z    +0.000, E1   +24.542, E3 +480374.211}
SPL {X  -162.820, Y  +606.285, Z    +0.000, E1   +24.533, E3 +480386.546}
SPL {X  -162.820, Y  +603.509, Z    +0.000, E1   +24.546, E3 +480399.084}
SPL {X  -162.820, Y  +600.818, Z    +0.000, E1   +24.590, E3 +480411.006}
SPL {X  -162.820, Y  +598.053, Z    +0.000, E1   +24.547, E3 +480423.989}
SPL {X  -162.820, Y  +595.188, Z    +0.000, E1   +24.538, E3 +480437.078}
SPL {X  -162.820, Y  +592.738, Z    +0.000, E1   +24.551, E3 +480448.126}
SPL {X  -162.820, Y  +590.118, Z    +0.000, E1   +24.544, E3 +480460.185}
SPL {X  -162.820, Y  +587.204, Z    +0.000, E1   +24.592, E3 +480473.062}
SPL {X  -162.820, Y  +584.766, Z    +0.000, E1   +24.499, E3 +480484.895}
SPL {X  -162.820, Y  +581.896, Z    +0.000, E1   +24.528, E3 +480497.837}
SPL {X  -162.820, Y  +579.244, Z    +0.000, E1   +24.610, E3 +480509.181}
SPL {X  -162.820, Y  +576.848, Z    +0.000, E1   +24.543, E3 +480520.723}
SPL {X  -162.820, Y  +573.694, Z    +0.000, E1   +24.535, E3 +480535.192}
SPL {X  -162.820, Y  +571.322, Z    +0.000, E1   +24.492, E3 +480546.226}
SPL {X  -162.820, Y  +568.309, Z    +0.000, E1   +24.589, E3 +480559.451}
SPL {X  -162.820, Y  +564.977, Z    +0.000, E1   +24.571, E3 +480574.624}
SPL {X  -162.820, Y  +562.356, Z    +0.000, E1   +24.575, E3 +480586.523}
SPL {X  -162.820, Y  +560.119, Z    +0.000, E1   +24.506, E3 +480597.211}
SPL {X  -162.820, Y  +558.093, Z    +0.000, E1   +24.537, E3 +480606.229}
SPL {X  -162.820, Y  +555.584, Z    +0.000, E1   +24.559, E3 +480617.541}
SPL {X  -162.820, Y  +552.169, Z    +0.000, E1   +24.581, E3 +480633.110}
SPL {X  -162.820, Y  +548.172, Z    +0.000, E1   +24.564, E3 +480651.458}
SPL {X  -162.820, Y  +544.025, Z    +0.000, E1   +24.611, E3 +480670.012}
SPL {X  -162.820, Y  +540.573, Z    +0.000, E1   +24.503, E3 +480686.467}
SPL {X  -162.820, Y  +538.106, Z    +0.000, E1   +24.553, E3 +480697.221}
SPL {X  -162.820, Y  +536.451, Z    +0.000, E1   +24.519, E3 +480705.039}
SPL {X  -162.820, Y  +534.025, Z    +0.000, E1   +24.589, E3 +480715.639}
SPL {X  -162.820, Y  +531.527, Z    +0.000, E1   +24.582, E3 +480727.024}
SPL {X  -162.820, Y  +529.165, Z    +0.000, E1   +24.521, E3 +480738.273}
SPL {X  -162.820, Y  +525.802, Z    +0.000, E1   +24.585, E3 +480753.293}
SPL {X  -162.820, Y  +521.731, Z    +0.000, E1   +24.542, E3 +480772.229}
SPL {X  -162.820, Y  +518.185, Z    +0.000, E1   +24.561, E3 +480788.101}
SPL {X  -162.820, Y  +508.728, Z    +0.000, E1   +28.484, E3 +480798.641}
SPL {X  -162.820, Y  +500.664, Z    +0.000, E1   +31.476, E3 +480807.305}
SPL {X  -162.820, Y  +499.290, Z    +0.000, E1   +30.657, E3 +480817.587}
SPL {X  -162.820, Y  +497.700, Z    +0.000, E1   +29.785, E3 +480829.202}
SPL {X  -162.820, Y  +495.915, Z    +0.000, E1   +28.861, E3 +480842.295}
SPL {X  -162.820, Y  +494.678, Z    +0.000, E1   +27.647, E3 +480855.640}
SPL {X  -162.820, Y  +493.757, Z    +0.000, E1   +26.462, E3 +480868.000}
SPL {X  -162.820, Y  +491.420, Z    +0.000, E1   +25.780, E3 +480883.262}
SPL {X  -162.820, Y  +487.351, Z    +0.000, E1   +25.663, E3 +480901.778}
SPL {X  -162.820, Y  +484.247, Z    +0.000, E1   +25.651, E3 +480915.104}
SPL {X  -162.820, Y  +482.092, Z    +0.000, E1   +25.593, E3 +480924.931}
SPL {X  -162.820, Y  +479.578, Z    +0.000, E1   +25.634, E3 +480935.574}
SPL {X  -162.820, Y  +477.137, Z    +0.000, E1   +25.632, E3 +480946.153}
SPL {X  -162.820, Y  +473.770, Z    +0.000, E1   +25.664, E3 +480960.699}
SPL {X  -162.820, Y  +469.694, Z    +0.000, E1   +25.657, E3 +480978.430}
SPL {X  -162.820, Y  +465.727, Z    +0.000, E1   +25.676, E3 +480995.473}
SPL {X  -162.820, Y  +463.001, Z    +0.000, E1   +25.614, E3 +481007.589}
SPL {X  -162.820, Y  +459.882, Z    +0.000, E1   +25.674, E3 +481020.890}
SPL {X  -162.820, Y  +456.773, Z    +0.000, E1   +25.591, E3 +481034.836}
SPL {X  -162.820, Y  +454.429, Z    +0.000, E1   +25.642, E3 +481044.604}
SPL {X  -162.820, Y  +451.204, Z    +0.000, E1   +25.672, E3 +481058.631}
SPL {X  -162.820, Y  +447.822, Z    +0.000, E1   +25.664, E3 +481073.114}
SPL {X  -162.820, Y  +445.556, Z    +0.000, E1   +25.626, E3 +481083.245}
SPL {X  -162.820, Y  +443.328, Z    +0.000, E1   +25.642, E3 +481092.759}
SPL {X  -162.820, Y  +440.857, Z    +0.000, E1   +25.614, E3 +481103.794}
SPL {X  -162.820, Y  +437.636, Z    +0.000, E1   +25.597, E3 +481117.957}
SPL {X  -162.820, Y  +434.768, Z    +0.000, E1   +25.655, E3 +481129.859}
SPL {X  -162.820, Y  +431.823, Z    +0.000, E1   +25.651, E3 +481142.858}
SPL {X  -162.820, Y  +427.740, Z    +0.000, E1   +25.667, E3 +481160.486}
SPL {X  -162.820, Y  +423.655, Z    +0.000, E1   +25.628, E3 +481178.510}
SPL {X  -162.820, Y  +419.407, Z    +0.000, E1   +25.665, E3 +481196.703}
SPL {X  -162.820, Y  +415.900, Z    +0.000, E1   +25.638, E3 +481211.972}
SPL {X  -162.820, Y  +413.088, Z    +0.000, E1   +25.644, E3 +481224.128}
SPL {X  -162.820, Y  +410.320, Z    +0.000, E1   +25.604, E3 +481236.447}
SPL {X  -162.820, Y  +407.487, Z    +0.000, E1   +25.617, E3 +481248.655}
SPL {X  -162.820, Y  +405.108, Z    +0.000, E1   +25.535, E3 +481259.623}
SPL {X  -162.820, Y  +401.373, Z    +0.000, E1   +25.736, E3 +481274.459}
SPL {X  -162.820, Y  +397.357, Z    +0.000, E1   +25.652, E3 +481292.529}
SPL {X  -162.820, Y  +393.659, Z    +0.000, E1   +25.666, E3 +481308.329}
SPL {X  -162.820, Y  +390.679, Z    +0.000, E1   +25.624, E3 +481321.573}
SPL {X  -162.820, Y  +387.939, Z    +0.000, E1   +25.627, E3 +481333.432}
SPL {X  -162.820, Y  +384.398, Z    +0.000, E1   +25.707, E3 +481348.330}
SPL {X  -162.820, Y  +380.448, Z    +0.000, E1   +25.674, E3 +481365.694}
SPL {X  -162.785, Y  +377.106, Z    +0.000, E1   +25.598, E3 +481380.638}
SPL {X  -162.709, Y  +374.484, Z    +0.000, E1   +25.711, E3 +481391.089}
SPL {X  -162.623, Y  +372.485, Z    +0.000, E1   +25.631, E3 +481400.369}
SPL {X  -162.487, Y  +370.088, Z    +0.000, E1   +25.525, E3 +481411.623}
SPL {X  -162.243, Y  +366.801, Z    +0.000, E1   +25.618, E3 +481425.264}
SPL {X  -161.977, Y  +363.953, Z    +0.000, E1   +25.528, E3 +481438.190}
SPL {X  -161.695, Y  +361.389, Z    +0.000, E1   +25.445, E3 +481450.006}
SPL {X  -161.364, Y  +358.774, Z    +0.000, E1   +25.454, E3 +481461.206}
SPL {X  -160.939, Y  +355.820, Z    +0.000, E1   +26.179, E3 +481468.424}
SPL {X  -155.035, Y  +330.756, Z    +0.000, E1   +37.918, E3 +481474.758}
SPL {X  -153.918, Y  +327.401, Z    +0.000, E1   +34.677, E3 +481510.059}
ENDSPLINE

SPLINE
SPL {X  -159.701, Y  +348.785, Z    +0.000, E1   +24.361, E3 +481517.539}
SPL {X  -162.442, Y  +369.407, Z    +0.000, E1   +11.234, E3 +481547.174}
SPL {X  -162.820, Y  +384.333, Z    +0.000, E1    +1.902, E3 +481548.380}
SPL {X  -162.820, Y  +389.940, Z    +0.000, E1    -2.281, E3 +481551.302}
SPL {X  -162.820, Y  +396.652, Z    +0.000, E1    -7.520, E3 +481550.881}
SPL {X  -162.820, Y  +406.605, Z    +0.000, E1   -16.760, E3 +481543.357}
SPL {X  -162.820, Y  +420.013, Z    +0.000, E1   -22.833, E3 +481571.478}
SPL {X  -162.820, Y  +442.075, Z    +0.000, E1   -31.090, E3 +481604.264}
ENDSPLINE

SPLINE
SPL {X  -162.820, Y  +436.949, Z    +0.000, E1   -25.871, E3 +481621.015}
ENDSPLINE

SPLINE
SPL {X  -162.820, Y  +439.120, Z    +0.000, E1   -25.352, E3 +481634.264}
SPL {X  -162.820, Y  +441.593, Z    +0.000, E1   -25.391, E3 +481644.816}
SPL {X  -162.820, Y  +444.317, Z    +0.000, E1   -25.492, E3 +481655.997}
SPL {X  -162.820, Y  +447.641, Z    +0.000, E1   -25.460, E3 +481670.932}
SPL {X  -162.820, Y  +451.939, Z    +0.000, E1   -25.468, E3 +481689.752}
SPL {X  -162.820, Y  +455.480, Z    +0.000, E1   -25.454, E3 +481705.164}
SPL {X  -162.820, Y  +458.079, Z    +0.000, E1   -25.369, E3 +481717.199}
SPL {X  -162.820, Y  +460.719, Z    +0.000, E1   -25.411, E3 +481728.457}
SPL {X  -162.820, Y  +463.419, Z    +0.000, E1   -25.510, E3 +481739.495}
SPL {X  -162.820, Y  +465.376, Z    +0.000, E1   -25.372, E3 +481749.083}
SPL {X  -162.820, Y  +467.440, Z    +0.000, E1   -25.427, E3 +481757.714}
SPL {X  -162.820, Y  +470.010, Z    +0.000, E1   -25.445, E3 +481768.919}
SPL {X  -162.820, Y  +473.445, Z    +0.000, E1   -25.493, E3 +481783.643}
SPL {X  -162.820, Y  +476.157, Z    +0.000, E1   -25.426, E3 +481795.858}
SPL {X  -162.820, Y  +478.461, Z    +0.000, E1   -25.410, E3 +481806.137}
SPL {X  -162.820, Y  +481.644, Z    +0.000, E1   -25.433, E3 +481820.084}
SPL {X  -162.820, Y  +486.042, Z    +0.000, E1   -25.483, E3 +481839.003}
SPL {X  -162.820, Y  +490.287, Z    +0.000, E1   -25.463, E3 +481857.721}
SPL {X  -162.820, Y  +493.705, Z    +0.000, E1   -25.443, E3 +481872.678}
SPL {X  -162.820, Y  +497.247, Z    +0.000, E1   -25.470, E3 +481888.140}
SPL {X  -162.820, Y  +501.343, Z    +0.000, E1   -25.435, E3 +481906.339}
SPL {X  -162.820, Y  +505.370, Z    +0.000, E1   -25.456, E3 +481923.803}
SPL {X  -162.820, Y  +509.412, Z    +0.000, E1   -25.458, E3 +481941.525}
SPL {X  -162.820, Y  +512.406, Z    +0.000, E1   -25.425, E3 +481954.682}
SPL {X  -162.820, Y  +515.039, Z    +0.000, E1   -25.452, E3 +481966.092}
SPL {X  -162.820, Y  +518.350, Z    +0.000, E1   -25.425, E3 +481980.842}
SPL {X  -162.820, Y  +521.486, Z    +0.000, E1   -25.382, E3 +481994.869}
SPL {X  -162.820, Y  +524.180, Z    +0.000, E1   -25.495, E3 +482005.742}
SPL {X  -162.820, Y  +527.020, Z    +0.000, E1   -25.477, E3 +482018.434}
SPL {X  -162.820, Y  +530.432, Z    +0.000, E1   -25.477, E3 +482033.301}
SPL {X  -162.820, Y  +534.051, Z    +0.000, E1   -25.484, E3 +482049.178}
SPL {X  -162.820, Y  +537.226, Z    +0.000, E1   -25.378, E3 +482063.747}
SPL {X  -162.820, Y  +539.521, Z    +0.000, E1   -25.386, E3 +482073.706}
SPL {X  -162.820, Y  +542.667, Z    +0.000, E1   -25.474, E3 +482087.031}
SPL {X  -162.820, Y  +546.125, Z    +0.000, E1   -25.505, E3 +482101.755}
SPL {X  -162.820, Y  +549.578, Z    +0.000, E1   -25.462, E3 +482117.379}
SPL {X  -162.820, Y  +553.157, Z    +0.000, E1   -25.443, E3 +482133.043}
SPL {X  -162.820, Y  +556.150, Z    +0.000, E1   -25.445, E3 +482146.133}
SPL {X  -162.820, Y  +559.215, Z    +0.000, E1   -25.460, E3 +482159.434}
SPL {X  -162.820, Y  +562.125, Z    +0.000, E1   -25.434, E3 +482172.355}
SPL {X  -162.820, Y  +564.880, Z    +0.000, E1   -25.448, E3 +482184.309}
SPL {X  -162.820, Y  +568.326, Z    +0.000, E1   -25.470, E3 +482199.368}
SPL {X  -162.820, Y  +572.331, Z    +0.000, E1   -25.489, E3 +482216.744}
SPL {X  -162.820, Y  +576.045, Z    +0.000, E1   -25.412, E3 +482233.552}
SPL {X  -162.820, Y  +580.038, Z    +0.000, E1   -25.473, E3 +482250.647}
SPL {X  -162.820, Y  +583.044, Z    +0.000, E1   -25.450, E3 +482263.770}
SPL {X  -162.820, Y  +585.512, Z    +0.000, E1   -25.448, E3 +482274.665}
SPL {X  -162.820, Y  +588.371, Z    +0.000, E1   -25.460, E3 +482287.051}
SPL {X  -162.820, Y  +590.476, Z    +0.000, E1   -25.398, E3 +482296.693}
SPL {X  -162.820, Y  +593.604, Z    +0.000, E1   -25.477, E3 +482309.971}
SPL {X  -162.820, Y  +596.868, Z    +0.000, E1   -25.461, E3 +482324.236}
SPL {X  -162.820, Y  +600.326, Z    +0.000, E1   -25.438, E3 +482339.757}
SPL {X  -162.820, Y  +604.526, Z    +0.000, E1   -25.502, E3 +482357.581}
SPL {X  -162.820, Y  +607.811, Z    +0.000, E1   -25.507, E3 +482371.795}
SPL {X  -162.820, Y  +610.517, Z    +0.000, E1   -25.412, E3 +482384.358}
SPL {X  -162.820, Y  +613.762, Z    +0.000, E1   -25.472, E3 +482398.165}
SPL {X  -162.820, Y  +617.275, Z    +0.000, E1   -25.466, E3 +482413.603}
SPL {X  -162.820, Y  +621.264, Z    +0.000, E1   -25.514, E3 +482430.765}
SPL {X  -162.820, Y  +624.430, Z    +0.000, E1   -25.475, E3 +482444.696}
SPL {X  -162.820, Y  +626.570, Z    +0.000, E1   -25.441, E3 +482454.296}
SPL {X  -162.820, Y  +628.902, Z    +0.000, E1   -25.449, E3 +482464.476}
SPL {X  -162.820, Y  +631.177, Z    +0.000, E1   -25.467, E3 +482474.308}
SPL {X  -162.820, Y  +633.994, Z    +0.000, E1   -25.503, E3 +482486.354}
SPL {X  -162.820, Y  +637.619, Z    +0.000, E1   -25.497, E3 +482502.414}
SPL {X  -162.820, Y  +640.803, Z    +0.000, E1   -25.462, E3 +482516.377}
SPL {X  -162.820, Y  +643.028, Z    +0.000, E1   -25.494, E3 +482525.886}
SPL {X  -162.820, Y  +646.519, Z    +0.000, E1   -25.551, E3 +482540.868}
SPL {X  -162.820, Y  +649.837, Z    +0.000, E1   -25.446, E3 +482555.993}
SPL {X  -162.820, Y  +652.810, Z    +0.000, E1   -25.497, E3 +482568.635}
SPL {X  -162.820, Y  +655.214, Z    +0.000, E1   -25.485, E3 +482579.138}
SPL {X  -162.820, Y  +657.616, Z    +0.000, E1   -25.511, E3 +482589.492}
SPL {X  -162.820, Y  +660.851, Z    +0.000, E1   -25.520, E3 +482603.635}
SPL {X  -162.820, Y  +663.853, Z    +0.000, E1   -25.496, E3 +482616.816}
SPL {X  -162.820, Y  +666.096, Z    +0.000, E1   -25.408, E3 +482627.283}
SPL {X  -162.820, Y  +668.238, Z    +0.000, E1   -25.482, E3 +482636.100}
SPL {X  -162.820, Y  +671.102, Z    +0.000, E1   -25.514, E3 +482648.439}
SPL {X  -162.820, Y  +673.648, Z    +0.000, E1   -25.431, E3 +482660.106}
SPL {X  -162.796, Y  +676.319, Z    +0.000, E1   -25.526, E3 +482671.116}
SPL {X  -162.707, Y  +679.552, Z    +0.000, E1   -25.443, E3 +482685.990}
SPL {X  -162.545, Y  +682.952, Z    +0.000, E1   -25.510, E3 +482700.223}
SPL {X  -162.381, Y  +685.455, Z    +0.000, E1   -25.410, E3 +482711.910}
SPL {X  -162.102, Y  +688.774, Z    +0.000, E1   -25.417, E3 +482726.524}
SPL {X  -161.778, Y  +691.887, Z    +0.000, E1   -25.301, E3 +482740.826}
SPL {X  -161.319, Y  +695.558, Z    +0.000, E1   -25.832, E3 +482752.780}
SPL {X  -157.976, Y  +712.921, Z    +0.000, E1   -33.197, E3 +482766.171}
ENDSPLINE

SPLINE
SPL {X  -160.738, Y  +699.453, Z    +0.000, E1   -21.994, E3 +482803.799}
SPL {X  -160.945, Y  +698.140, Z    +0.000, E1   -18.412, E3 +482846.038}
SPL {X  -162.497, Y  +683.755, Z    +0.000, E1   -10.754, E3 +482840.182}
SPL {X  -162.819, Y  +673.996, Z    +0.000, E1    -4.745, E3 +482839.783}
ENDSPLINE

SPLINE
SPL {X  -162.791, Y  +676.574, Z    +0.000, E1    -6.127, E3 +482852.471}
ENDSPLINE

SPLINE
SPL {X  -162.820, Y  +667.935, Z    +0.000, E1    -0.509, E3 +482842.557}
SPL {X  -162.820, Y  +662.949, Z    +0.000, E1    +3.113, E3 +482840.676}
SPL {X  -162.820, Y  +658.484, Z    +0.000, E1    +6.336, E3 +482847.821}
SPL {X  -162.820, Y  +640.102, Z    +0.000, E1   +22.409, E3 +482842.560}
SPL {X  -162.820, Y  +633.503, Z    +0.000, E1   +21.975, E3 +482874.796}
SPL {X  -162.820, Y  +611.299, Z    +0.000, E1   +31.088, E3 +482902.909}
ENDSPLINE

SPLINE
SPL {X  -162.820, Y  +618.877, Z    +0.000, E1   +25.259, E3 +482914.403}
ENDSPLINE

SPLINE
SPL {X  -162.820, Y  +617.582, Z    +0.000, E1   +24.552, E3 +482925.780}
SPL {X  -162.820, Y  +614.716, Z    +0.000, E1   +24.535, E3 +482938.991}
SPL {X  -162.820, Y  +611.754, Z    +0.000, E1   +24.563, E3 +482952.280}
SPL {X  -162.820, Y  +608.970, Z    +0.000, E1   +24.542, E3 +482965.120}
SPL {X  -162.820, Y  +606.285, Z    +0.000, E1   +24.533, E3 +482977.455}
SPL {X  -162.820, Y  +603.509, Z    +0.000, E1   +24.546, E3 +482989.993}
SPL {X  -162.820, Y  +600.230, Z    +0.000, E1   +24.589, E3 +483004.737}
SPL {X  -162.820, Y  +597.446, Z    +0.000, E1   +24.542, E3 +483017.596}
SPL {X  -162.820, Y  +595.188, Z    +0.000, E1   +24.538, E3 +483027.987}
SPL {X  -162.820, Y  +591.955, Z    +0.000, E1   +24.571, E3 +483042.607}
SPL {X  -162.820, Y  +587.913, Z    +0.000, E1   +24.604, E3 +483060.825}
SPL {X  -162.820, Y  +584.193, Z    +0.000, E1   +24.484, E3 +483078.681}
SPL {X  -162.820, Y  +580.163, Z    +0.000, E1   +24.634, E3 +483095.916}
SPL {X  -162.820, Y  +576.848, Z    +0.000, E1   +24.543, E3 +483111.632}
SPL {X  -162.820, Y  +574.433, Z    +0.000, E1   +24.551, E3 +483122.462}
SPL {X  -162.820, Y  +572.074, Z    +0.000, E1   +24.505, E3 +483133.734}
SPL {X  -162.820, Y  +568.309, Z    +0.000, E1   +24.589, E3 +483150.360}
SPL {X  -162.820, Y  +564.977, Z    +0.000, E1   +24.571, E3 +483165.533}
SPL {X  -162.820, Y  +562.356, Z    +0.000, E1   +24.575, E3 +483177.432}
SPL {X  -162.820, Y  +558.990, Z    +0.000, E1   +24.558, E3 +483193.082}
SPL {X  -162.820, Y  +555.584, Z    +0.000, E1   +24.559, E3 +483208.451}
SPL {X  -162.820, Y  +552.867, Z    +0.000, E1   +24.583, E3 +483220.646}
SPL {X  -162.820, Y  +549.589, Z    +0.000, E1   +24.547, E3 +483236.012}
SPL {X  -162.820, Y  +545.742, Z    +0.000, E1   +24.577, E3 +483253.299}
SPL {X  -162.820, Y  +542.142, Z    +0.000, E1   +24.582, E3 +483269.652}
SPL {X  -162.820, Y  +538.903, Z    +0.000, E1   +24.519, E3 +483284.868}
SPL {X  -162.820, Y  +536.451, Z    +0.000, E1   +24.519, E3 +483295.948}
SPL {X  -162.820, Y  +534.025, Z    +0.000, E1   +24.589, E3 +483306.548}
SPL {X  -162.820, Y  +531.527, Z    +0.000, E1   +24.582, E3 +483317.933}
SPL {X  -162.820, Y  +529.165, Z    +0.000, E1   +24.521, E3 +483329.182}
SPL {X  -162.820, Y  +525.802, Z    +0.000, E1   +24.585, E3 +483344.202}
SPL {X  -162.820, Y  +521.731, Z    +0.000, E1   +24.542, E3 +483363.138}
SPL {X  -162.820, Y  +518.185, Z    +0.000, E1   +24.561, E3 +483379.010}
SPL {X  -162.820, Y  +508.728, Z    +0.000, E1   +28.484, E3 +483389.550}
SPL {X  -162.820, Y  +500.664, Z    +0.000, E1   +31.476, E3 +483398.214}
SPL {X  -162.820, Y  +499.290, Z    +0.000, E1   +30.657, E3 +483408.496}
SPL {X  -162.820, Y  +497.700, Z    +0.000, E1   +29.785, E3 +483420.111}
SPL {X  -162.820, Y  +495.915, Z    +0.000, E1   +28.861, E3 +483433.204}
SPL {X  -162.820, Y  +494.678, Z    +0.000, E1   +27.647, E3 +483446.549}
SPL {X  -162.820, Y  +493.757, Z    +0.000, E1   +26.462, E3 +483458.909}
SPL {X  -162.820, Y  +491.420, Z    +0.000, E1   +25.780, E3 +483474.171}
SPL {X  -162.820, Y  +487.351, Z    +0.000, E1   +25.663, E3 +483492.687}
SPL {X  -162.820, Y  +484.247, Z    +0.000, E1   +25.651, E3 +483506.013}
SPL {X  -162.820, Y  +482.092, Z    +0.000, E1   +25.593, E3 +483515.840}
SPL {X  -162.820, Y  +479.578, Z    +0.000, E1   +25.634, E3 +483526.483}
SPL {X  -162.820, Y  +477.137, Z    +0.000, E1   +25.632, E3 +483537.062}
SPL {X  -162.820, Y  +473.770, Z    +0.000, E1   +25.664, E3 +483551.608}
SPL {X  -162.820, Y  +469.694, Z    +0.000, E1   +25.657, E3 +483569.339}
SPL {X  -162.820, Y  +465.727, Z    +0.000, E1   +25.676, E3 +483586.382}
SPL {X  -162.820, Y  +461.675, Z    +0.000, E1   +25.655, E3 +483604.189}
SPL {X  -162.820, Y  +457.479, Z    +0.000, E1   +25.656, E3 +483622.368}
SPL {X  -162.820, Y  +453.678, Z    +0.000, E1   +25.652, E3 +483638.821}
SPL {X  -162.820, Y  +450.466, Z    +0.000, E1   +25.644, E3 +483652.766}
SPL {X  -162.820, Y  +447.822, Z    +0.000, E1   +25.664, E3 +483664.023}
SPL {X  -162.820, Y  +444.499, Z    +0.000, E1   +25.673, E3 +483678.594}
SPL {X  -162.820, Y  +440.857, Z    +0.000, E1   +25.614, E3 +483694.703}
SPL {X  -162.820, Y  +438.582, Z    +0.000, E1   +25.544, E3 +483705.022}
SPL {X  -162.820, Y  +435.635, Z    +0.000, E1   +25.661, E3 +483717.118}
SPL {X  -162.820, Y  +431.823, Z    +0.000, E1   +25.651, E3 +483733.767}
SPL {X  -162.820, Y  +427.740, Z    +0.000, E1   +25.667, E3 +483751.395}
SPL {X  -162.820, Y  +423.655, Z    +0.000, E1   +25.628, E3 +483769.419}
SPL {X  -162.820, Y  +419.407, Z    +0.000, E1   +25.665, E3 +483787.612}
SPL {X  -162.820, Y  +415.900, Z    +0.000, E1   +25.638, E3 +483802.881}
SPL {X  -162.820, Y  +413.088, Z    +0.000, E1   +25.644, E3 +483815.037}
SPL {X  -162.820, Y  +410.320, Z    +0.000, E1   +25.604, E3 +483827.356}
SPL {X  -162.820, Y  +407.487, Z    +0.000, E1   +25.617, E3 +483839.564}
SPL {X  -162.820, Y  +405.108, Z    +0.000, E1   +25.535, E3 +483850.532}
SPL {X  -162.820, Y  +401.373, Z    +0.000, E1   +25.736, E3 +483865.368}
SPL {X  -162.820, Y  +397.357, Z    +0.000, E1   +25.652, E3 +483883.438}
SPL {X  -162.820, Y  +393.659, Z    +0.000, E1   +25.666, E3 +483899.238}
SPL {X  -162.820, Y  +390.679, Z    +0.000, E1   +25.624, E3 +483912.482}
SPL {X  -162.820, Y  +387.939, Z    +0.000, E1   +25.627, E3 +483924.341}
SPL {X  -162.820, Y  +384.398, Z    +0.000, E1   +25.707, E3 +483939.239}
SPL {X  -162.820, Y  +380.448, Z    +0.000, E1   +25.674, E3 +483956.603}
SPL {X  -162.785, Y  +377.106, Z    +0.000, E1   +25.598, E3 +483971.547}
SPL {X  -162.709, Y  +374.484, Z    +0.000, E1   +25.711, E3 +483981.998}
SPL {X  -162.623, Y  +372.485, Z    +0.000, E1   +25.631, E3 +483991.278}
SPL {X  -162.487, Y  +370.088, Z    +0.000, E1   +25.525, E3 +484002.532}
SPL {X  -162.243, Y  +366.801, Z    +0.000, E1   +25.618, E3 +484016.173}
SPL {X  -161.882, Y  +363.046, Z    +0.000, E1   +25.550, E3 +484033.056}
SPL {X  -161.454, Y  +359.455, Z    +0.000, E1   +25.428, E3 +484049.451}
SPL {X  -160.939, Y  +355.820, Z    +0.000, E1   +26.179, E3 +484059.333}
SPL {X  -154.424, Y  +328.890, Z    +0.000, E1   +36.591, E3 +484080.166}
ENDSPLINE

SPLINE
SPL {X  -159.701, Y  +348.785, Z    +0.000, E1   +24.361, E3 +484108.449}
SPL {X  -162.442, Y  +369.407, Z    +0.000, E1   +11.234, E3 +484138.084}
SPL {X  -162.820, Y  +384.333, Z    +0.000, E1    +1.902, E3 +484139.290}
SPL {X  -162.820, Y  +389.940, Z    +0.000, E1    -2.281, E3 +484142.211}
SPL {X  -162.820, Y  +396.652, Z    +0.000, E1    -7.520, E3 +484141.790}
SPL {X  -162.820, Y  +406.605, Z    +0.000, E1   -16.760, E3 +484134.267}
SPL {X  -162.820, Y  +420.013, Z    +0.000, E1   -22.833, E3 +484162.387}
SPL {X  -162.820, Y  +442.075, Z    +0.000, E1   -31.090, E3 +484195.173}
ENDSPLINE

SPLINE
SPL {X  -162.820, Y  +436.949, Z    +0.000, E1   -25.871, E3 +484211.924}
ENDSPLINE

SPLINE
SPL {X  -162.820, Y  +439.120, Z    +0.000, E1   -25.352, E3 +484225.173}
SPL {X  -162.820, Y  +441.593, Z    +0.000, E1   -25.391, E3 +484235.725}
SPL {X  -162.820, Y  +444.317, Z    +0.000, E1   -25.492, E3 +484246.906}
SPL {X  -162.820, Y  +447.641, Z    +0.000, E1   -25.460, E3 +484261.841}
SPL {X  -162.820, Y  +451.939, Z    +0.000, E1   -25.468, E3 +484280.662}
SPL {X  -162.820, Y  +455.480, Z    +0.000, E1   -25.454, E3 +484296.073}
SPL {X  -162.820, Y  +458.079, Z    +0.000, E1   -25.369, E3 +484308.108}
SPL {X  -162.820, Y  +460.719, Z    +0.000, E1   -25.411, E3 +484319.366}
SPL {X  -162.820, Y  +463.419, Z    +0.000, E1   -25.510, E3 +484330.404}
SPL {X  -162.820, Y  +466.458, Z    +0.000, E1   -25.433, E3 +484344.460}
SPL {X  -162.820, Y  +470.010, Z    +0.000, E1   -25.445, E3 +484359.828}
SPL {X  -162.820, Y  +473.445, Z    +0.000, E1   -25.493, E3 +484374.552}
SPL {X  -162.820, Y  +476.157, Z    +0.000, E1   -25.426, E3 +484386.767}
SPL {X  -162.820, Y  +478.461, Z    +0.000, E1   -25.410, E3 +484397.046}
SPL {X  -162.820, Y  +481.644, Z    +0.000, E1   -25.433, E3 +484410.993}
SPL {X  -162.820, Y  +486.042, Z    +0.000, E1   -25.483, E3 +484429.912}
SPL {X  -162.820, Y  +490.287, Z    +0.000, E1   -25.463, E3 +484448.630}
SPL {X  -162.820, Y  +494.454, Z    +0.000, E1   -25.465, E3 +484466.862}
SPL {X  -162.820, Y  +497.898, Z    +0.000, E1   -25.452, E3 +484481.884}
SPL {X  -162.820, Y  +501.343, Z    +0.000, E1   -25.435, E3 +484497.248}
SPL {X  -162.820, Y  +505.370, Z    +0.000, E1   -25.456, E3 +484514.712}
SPL {X  -162.820, Y  +508.346, Z    +0.000, E1   -25.444, E3 +484527.659}
SPL {X  -162.820, Y  +511.422, Z    +0.000, E1   -25.445, E3 +484541.320}
SPL {X  -162.820, Y  +515.039, Z    +0.000, E1   -25.452, E3 +484557.001}
SPL {X  -162.820, Y  +517.481, Z    +0.000, E1   -25.432, E3 +484567.736}
SPL {X  -162.820, Y  +519.134, Z    +0.000, E1   -25.366, E3 +484575.482}
SPL {X  -162.820, Y  +521.486, Z    +0.000, E1   -25.382, E3 +484585.778}
SPL {X  -162.820, Y  +525.073, Z    +0.000, E1   -25.512, E3 +484600.584}
SPL {X  -162.820, Y  +527.738, Z    +0.000, E1   -25.438, E3 +484612.632}
SPL {X  -162.820, Y  +530.432, Z    +0.000, E1   -25.477, E3 +484624.210}
SPL {X  -162.820, Y  +534.051, Z    +0.000, E1   -25.484, E3 +484640.087}
SPL {X  -162.820, Y  +537.226, Z    +0.000, E1   -25.378, E3 +484654.656}
SPL {X  -162.820, Y  +540.345, Z    +0.000, E1   -25.451, E3 +484667.837}
SPL {X  -162.820, Y  +543.279, Z    +0.000, E1   -25.419, E3 +484680.870}
SPL {X  -162.820, Y  +546.125, Z    +0.000, E1   -25.505, E3 +484692.664}
SPL {X  -162.820, Y  +549.578, Z    +0.000, E1   -25.462, E3 +484708.289}
SPL {X  -162.820, Y  +553.157, Z    +0.000, E1   -25.443, E3 +484723.952}
SPL {X  -162.820, Y  +556.150, Z    +0.000, E1   -25.445, E3 +484737.042}
SPL {X  -162.820, Y  +559.215, Z    +0.000, E1   -25.460, E3 +484750.343}
SPL {X  -162.820, Y  +562.125, Z    +0.000, E1   -25.434, E3 +484763.264}
SPL {X  -162.820, Y  +564.880, Z    +0.000, E1   -25.448, E3 +484775.218}
SPL {X  -162.820, Y  +568.326, Z    +0.000, E1   -25.470, E3 +484790.277}
SPL {X  -162.820, Y  +571.303, Z    +0.000, E1   -25.427, E3 +484803.450}
SPL {X  -162.820, Y  +574.067, Z    +0.000, E1   -25.459, E3 +484815.389}
SPL {X  -162.820, Y  +576.597, Z    +0.000, E1   -25.400, E3 +484826.860}
SPL {X  -162.820, Y  +578.977, Z    +0.000, E1   -25.460, E3 +484836.793}
SPL {X  -162.820, Y  +581.995, Z    +0.000, E1   -25.468, E3 +484850.151}
SPL {X  -162.820, Y  +585.512, Z    +0.000, E1   -25.448, E3 +484865.575}
SPL {X  -162.820, Y  +588.371, Z    +0.000, E1   -25.460, E3 +484877.961}
SPL {X  -162.820, Y  +591.246, Z    +0.000, E1   -25.415, E3 +484890.980}
SPL {X  -162.820, Y  +594.339, Z    +0.000, E1   -25.487, E3 +484903.882}
SPL {X  -162.820, Y  +596.868, Z    +0.000, E1   -25.461, E3 +484915.145}
SPL {X  -162.820, Y  +600.326, Z    +0.000, E1   -25.438, E3 +484930.667}
SPL {X  -162.820, Y  +604.526, Z    +0.000, E1   -25.502, E3 +484948.490}
SPL {X  -162.820, Y  +607.811, Z    +0.000, E1   -25.507, E3 +484962.704}
SPL {X  -162.820, Y  +610.517, Z    +0.000, E1   -25.412, E3 +484975.267}
SPL {X  -162.820, Y  +613.762, Z    +0.000, E1   -25.472, E3 +484989.074}
SPL {X  -162.820, Y  +617.275, Z    +0.000, E1   -25.466, E3 +485004.513}
SPL {X  -162.820, Y  +621.264, Z    +0.000, E1   -25.514, E3 +485021.674}
SPL {X  -162.820, Y  +624.430, Z    +0.000, E1   -25.475, E3 +485035.605}
SPL {X  -162.820, Y  +626.570, Z    +0.000, E1   -25.441, E3 +485045.205}
SPL {X  -162.820, Y  +628.902, Z    +0.000, E1   -25.449, E3 +485055.385}
SPL {X  -162.820, Y  +631.177, Z    +0.000, E1   -25.467, E3 +485065.217}
SPL {X  -162.820, Y  +633.994, Z    +0.000, E1   -25.503, E3 +485077.263}
SPL {X  -162.820, Y  +636.469, Z    +0.000, E1   -25.465, E3 +485088.307}
SPL {X  -162.820, Y  +638.486, Z    +0.000, E1   -25.456, E3 +485097.224}
SPL {X  -162.820, Y  +640.803, Z    +0.000, E1   -25.462, E3 +485107.286}
SPL {X  -162.820, Y  +643.028, Z    +0.000, E1   -25.494, E3 +485116.795}
SPL {X  -162.820, Y  +645.694, Z    +0.000, E1   -25.540, E3 +485128.083}
SPL {X  -162.820, Y  +649.102, Z    +0.000, E1   -25.495, E3 +485143.511}
SPL {X  -162.820, Y  +652.810, Z    +0.000, E1   -25.497, E3 +485159.544}
SPL {X  -162.820, Y  +655.214, Z    +0.000, E1   -25.485, E3 +485170.047}
SPL {X  -162.820, Y  +657.616, Z    +0.000, E1   -25.511, E3 +485180.401}
SPL {X  -162.820, Y  +660.007, Z    +0.000, E1   -25.550, E3 +485190.463}
SPL {X  -162.820, Y  +662.980, Z    +0.000, E1   -25.505, E3 +485204.021}
SPL {X  -162.820, Y  +666.096, Z    +0.000, E1   -25.408, E3 +485218.193}
SPL {X  -162.820, Y  +669.195, Z    +0.000, E1   -25.525, E3 +485231.030}
SPL {X  -162.820, Y  +672.979, Z    +0.000, E1   -25.478, E3 +485247.880}
SPL {X  -162.796, Y  +676.319, Z    +0.000, E1   -25.526, E3 +485262.025}
SPL {X  -162.739, Y  +678.625, Z    +0.000, E1   -25.423, E3 +485272.816}
SPL {X  -162.669, Y  +680.515, Z    +0.000, E1   -25.398, E3 +485281.270}
SPL {X  -162.545, Y  +682.952, Z    +0.000, E1   -25.510, E3 +485291.132}
SPL {X  -162.381, Y  +685.455, Z    +0.000, E1   -25.410, E3 +485302.819}
SPL {X  -162.194, Y  +687.760, Z    +0.000, E1   -25.360, E3 +485313.255}
SPL {X  -161.866, Y  +691.104, Z    +0.000, E1   -25.383, E3 +485327.887}
SPL {X  -161.024, Y  +697.619, Z    +0.000, E1   -26.780, E3 +485345.117}
SPL {X  -157.189, Y  +715.948, Z    +0.000, E1   -34.218, E3 +485360.036}
ENDSPLINE

SPLINE
SPL {X  -157.848, Y  +713.428, Z    +0.000, E1   -28.857, E3 +485394.175}
SPL {X  -161.035, Y  +697.541, Z    +0.000, E1   -20.899, E3 +485394.694}
ENDSPLINE

SPLINE
SPL {X  -160.945, Y  +698.140, Z    +0.000, E1   -18.412, E3 +485436.947}
ENDSPLINE

SPLINE
SPL {X  -162.497, Y  +683.755, Z    +0.000, E1   -10.754, E3 +485431.091}
SPL {X  -162.819, Y  +673.996, Z    +0.000, E1    -4.745, E3 +485430.692}
ENDSPLINE

SPLINE
SPL {X  -162.791, Y  +676.574, Z    +0.000, E1    -6.127, E3 +485443.380}
ENDSPLINE

SPLINE
SPL {X  -162.820, Y  +667.935, Z    +0.000, E1    -0.509, E3 +485433.466}
SPL {X  -162.820, Y  +662.949, Z    +0.000, E1    +3.113, E3 +485431.585}
SPL {X  -162.820, Y  +658.484, Z    +0.000, E1    +6.336, E3 +485438.730}
SPL {X  -162.820, Y  +640.102, Z    +0.000, E1   +22.409, E3 +485433.469}
SPL {X  -162.820, Y  +633.503, Z    +0.000, E1   +21.975, E3 +485465.705}
SPL {X  -162.820, Y  +611.299, Z    +0.000, E1   +31.088, E3 +485493.818}
ENDSPLINE

SPLINE
SPL {X  -162.820, Y  +618.877, Z    +0.000, E1   +25.259, E3 +485505.312}
ENDSPLINE

SPLINE
SPL {X  -162.820, Y  +617.582, Z    +0.000, E1   +24.552, E3 +485516.689}
SPL {X  -162.820, Y  +614.716, Z    +0.000, E1   +24.535, E3 +485529.900}
SPL {X  -162.820, Y  +611.754, Z    +0.000, E1   +24.563, E3 +485543.189}
SPL {X  -162.820, Y  +608.970, Z    +0.000, E1   +24.542, E3 +485556.029}
SPL {X  -162.820, Y  +606.285, Z    +0.000, E1   +24.533, E3 +485568.364}
SPL {X  -162.820, Y  +603.509, Z    +0.000, E1   +24.546, E3 +485580.902}
SPL {X  -162.820, Y  +600.230, Z    +0.000, E1   +24.589, E3 +485595.646}
SPL {X  -162.820, Y  +597.446, Z    +0.000, E1   +24.542, E3 +485608.505}
SPL {X  -162.820, Y  +595.188, Z    +0.000, E1   +24.538, E3 +485618.896}
SPL {X  -162.820, Y  +591.955, Z    +0.000, E1   +24.571, E3 +485633.516}
SPL {X  -162.820, Y  +587.913, Z    +0.000, E1   +24.604, E3 +485651.734}
SPL {X  -162.820, Y  +584.193, Z    +0.000, E1   +24.484, E3 +485669.590}
SPL {X  -162.820, Y  +581.176, Z    +0.000, E1   +24.592, E3 +485682.352}
SPL {X  -162.820, Y  +578.588, Z    +0.000, E1   +24.598, E3 +485694.207}
SPL {X  -162.820, Y  +576.196, Z    +0.000, E1   +24.519, E3 +485705.590}
SPL {X  -162.820, Y  +573.694, Z    +0.000, E1   +24.535, E3 +485717.010}
SPL {X  -162.820, Y  +570.310, Z    +0.000, E1   +24.556, E3 +485732.327}
SPL {X  -162.820, Y  +567.494, Z    +0.000, E1   +24.547, E3 +485745.112}
SPL {X  -162.820, Y  +564.977, Z    +0.000, E1   +24.571, E3 +485756.442}
SPL {X  -162.820, Y  +562.356, Z    +0.000, E1   +24.575, E3 +485768.341}
SPL {X  -162.820, Y  +558.990, Z    +0.000, E1   +24.558, E3 +485783.991}
SPL {X  -162.820, Y  +555.584, Z    +0.000, E1   +24.559, E3 +485799.360}
SPL {X  -162.820, Y  +552.169, Z    +0.000, E1   +24.581, E3 +485814.929}
SPL {X  -162.820, Y  +548.172, Z    +0.000, E1   +24.564, E3 +485833.276}
SPL {X  -162.820, Y  +544.025, Z    +0.000, E1   +24.611, E3 +485851.831}
SPL {X  -162.820, Y  +540.573, Z    +0.000, E1   +24.503, E3 +485868.285}
SPL {X  -162.820, Y  +537.211, Z    +0.000, E1   +24.561, E3 +485883.214}
SPL {X  -162.820, Y  +534.025, Z    +0.000, E1   +24.589, E3 +485897.457}
SPL {X  -162.820, Y  +531.527, Z    +0.000, E1   +24.582, E3 +485908.843}
SPL {X  -162.820, Y  +529.165, Z    +0.000, E1   +24.521, E3 +485920.091}
SPL {X  -162.820, Y  +526.822, Z    +0.000, E1   +24.559, E3 +485930.455}
SPL {X  -162.820, Y  +524.112, Z    +0.000, E1   +24.542, E3 +485943.072}
SPL {X  -162.820, Y  +521.048, Z    +0.000, E1   +24.515, E3 +485957.209}
SPL {X  -162.820, Y  +518.185, Z    +0.000, E1   +24.561, E3 +485969.920}
SPL {X  -162.820, Y  +508.728, Z    +0.000, E1   +28.484, E3 +485980.459}
SPL {X  -162.820, Y  +500.664, Z    +0.000, E1   +31.476, E3 +485989.123}
SPL {X  -162.820, Y  +499.290, Z    +0.000, E1   +30.657, E3 +485999.405}
SPL {X  -162.820, Y  +497.251, Z    +0.000, E1   +29.634, E3 +486013.881}
SPL {X  -162.820, Y  +495.647, Z    +0.000, E1   +28.606, E3 +486026.757}
SPL {X  -162.820, Y  +494.678, Z    +0.000, E1   +27.647, E3 +486037.458}
SPL {X  -162.820, Y  +493.757, Z    +0.000, E1   +26.462, E3 +486049.818}
SPL {X  -162.820, Y  +492.330, Z    +0.000, E1   +25.953, E3 +486059.572}
ENDSPLINE

SPLINE
SPL {X  -162.820, Y  +497.778, Z    +0.000, E1   +21.646, E3 +486068.488}
ENDSPLINE

